  Set speed (17.1 mm/s)
  Call Extruder(548.01735)
  MoveL 6241 to (555.94, 469.94, 108) mm, rotated rx 180 ry 0 rz 160 deg; joints [2.142, 70.681, -21.623, -151.69, 52.63, 161.895]
  Set speed (17.1 mm/s)
  Call Extruder(550.98604)
  MoveL 6242 to (556.35, 470.73, 108) mm, rotated rx 180 ry 0 rz 160 deg; joints [2.23, 70.775, -21.811, -151.55, 52.574, 161.774]
  Set speed (17.1 mm/s)
  Call Extruder(555.34472)
  MoveL 6243 to (556.95, 471.91, 108) mm, rotated rx 180 ry 0 rz 160 deg; joints [2.36, 70.91, -22.084, -151.344, 52.494, 161.596]
  Set speed (17.1 mm/s)
  Call Extruder(559.57401)
  MoveL 6244 to (557.5, 473.06, 108) mm, rotated rx -180 ry 0 rz 160 deg; joints [2.488, 71.037, -22.339, -151.143, 52.422, 161.425]
  Set speed (17.1 mm/s)
  Call Extruder(563.96084)
  MoveL 6245 to (558.05, 474.27, 108) mm, rotated rx -180 ry 0 rz 160 deg; joints [2.621, 71.165, -22.597, -150.936, 52.351, 161.248]
  Set speed (17.1 mm/s)
  Call Extruder(568.24026)
  MoveL 6246 to (558.56, 475.46, 108) mm, rotated rx 180 ry 0 rz 160 deg; joints [2.752, 71.285, -22.838, -150.733, 52.288, 161.078]
  Set speed (17.1 mm/s)
  Call Extruder(572.63486)
  MoveL 6247 to (559.07, 476.69, 108) mm, rotated rx 180 ry 0 rz 160 deg; joints [2.888, 71.406, -23.081, -150.525, 52.225, 160.903]
  Set speed (17.0 mm/s)
  Call Extruder(577.61580)
  MoveL 6248 to (559.6, 478.09, 108) mm, rotated rx 180 ry 0 rz 160 deg; joints [3.043, 71.535, -23.342, -150.289, 52.162, 160.707]
  Set speed (17.0 mm/s)
  Call Extruder(581.16765)
  MoveL 6249 to (559.96, 479.1, 108) mm, rotated rx 180 ry 0 rz 160 deg; joints [3.154, 71.626, -23.524, -150.121, 52.12, 160.569]
  Set speed (17.0 mm/s)
  Call Extruder(585.42677)
  MoveL 6250 to (560.37, 480.32, 108) mm, rotated rx -180 ry 0 rz 160 deg; joints [3.288, 71.728, -23.73, -149.92, 52.075, 160.404]
  Set speed (17.1 mm/s)
  Call Extruder(589.90951)
  MoveL 6251 to (560.78, 481.61, 108) mm, rotated rx -180 ry 0 rz 160 deg; joints [3.43, 71.835, -23.944, -149.709, 52.03, 160.232]
  Set speed (17.1 mm/s)
  Call Extruder(594.01666)
  MoveL 6252 to (561.12, 482.81, 108) mm, rotated rx 180 ry 0 rz 160 deg; joints [3.561, 71.925, -24.125, -149.516, 51.996, 160.077]
  Call Extruder(598.21491)
  MoveL 6253 to (561.46, 484.03, 108) mm, rotated rx 180 ry 0 rz 160 deg; joints [3.695, 72.016, -24.307, -149.32, 51.963, 159.919]
  Set speed (17.1 mm/s)
  Call Extruder(602.61345)
  MoveL 6254 to (561.77, 485.32, 108) mm, rotated rx -180 ry 0 rz 160 deg; joints [3.837, 72.104, -24.483, -149.115, 51.936, 159.758]
  Call Extruder(606.81186)
  MoveL 6255 to (562.06, 486.56, 108) mm, rotated rx -180 ry 0 rz 160 deg; joints [3.973, 72.186, -24.648, -148.92, 51.912, 159.604]
  Set speed (17.1 mm/s)
  Call Extruder(615.47372)
  MoveL 6256 to (562.56, 489.13, 108) mm, rotated rx 180 ry 0 rz 160 deg; joints [4.256, 72.337, -24.952, -148.522, 51.881, 159.296]
  Set speed (17.1 mm/s)
  Call Extruder(624.04952)
  MoveL 6257 to (562.96, 491.7, 108) mm, rotated rx 180 ry 0 rz 160 deg; joints [4.538, 72.468, -25.214, -148.133, 51.87, 159.001]
  Call Extruder(632.73234)
  MoveL 6258 to (563.25, 494.31, 108) mm, rotated rx 180 ry 0 rz 160 deg; joints [4.825, 72.581, -25.44, -147.745, 51.877, 158.714]
  Set speed (17.1 mm/s)
  Call Extruder(641.21506)
  MoveL 6259 to (563.42, 496.87, 108) mm, rotated rx 180 ry 0 rz 160 deg; joints [5.108, 72.671, -25.62, -147.373, 51.905, 158.447]
  Call Extruder(649.80353)
  MoveL 6260 to (563.5, 499.47, 108) mm, rotated rx 180 ry 0 rz 160 deg; joints [5.395, 72.741, -25.761, -147.004, 51.951, 158.189]
  Set speed (17.1 mm/s)
  Call Extruder(658.25838)
  MoveL 6261 to (563.47, 502.03, 108) mm, rotated rx 180 ry 0 rz 160 deg; joints [5.678, 72.79, -25.859, -146.649, 52.016, 157.949]
  Set speed (17.1 mm/s)
  Call Extruder(666.94750)
  MoveL 6262 to (563.33, 504.65, 108) mm, rotated rx 180 ry 0 rz 160 deg; joints [5.97, 72.82, -25.918, -146.293, 52.102, 157.718]
  Set speed (17.1 mm/s)
  Call Extruder(675.54081)
  MoveL 6263 to (563.09, 507.24, 108) mm, rotated rx 180 ry 0 rz 160 deg; joints [6.259, 72.827, -25.933, -145.952, 52.206, 157.505]
  Set speed (17.1 mm/s)
  Call Extruder(684.21964)
  MoveL 6264 to (562.73, 509.85, 108) mm, rotated rx -180 ry 0 rz 160 deg; joints [6.552, 72.813, -25.905, -145.617, 52.329, 157.306]
  Set speed (17.1 mm/s)
  Call Extruder(692.70275)
  MoveL 6265 to (562.29, 512.38, 108) mm, rotated rx -180 ry 0 rz 160 deg; joints [6.837, 72.779, -25.837, -145.3, 52.468, 157.128]
  Set speed (17.1 mm/s)
  Call Extruder(701.33186)
  MoveL 6266 to (561.72, 514.93, 108) mm, rotated rx 180 ry 0 rz 160 deg; joints [7.126, 72.723, -25.725, -144.989, 52.627, 156.965]
  Set speed (17.1 mm/s)
  Call Extruder(705.59645)
  MoveL 6267 to (561.4, 516.17, 108) mm, rotated rx 180 ry 0 rz 160 deg; joints [7.268, 72.686, -25.651, -144.841, 52.713, 156.892]
  Set speed (17.1 mm/s)
  Call Extruder(709.78855)
  MoveL 6268 to (561.07, 517.4, 108) mm, rotated rx -180 ry 0 rz 160 deg; joints [7.408, 72.648, -25.574, -144.696, 52.799, 156.822]
  Call Extruder(714.24503)
  MoveL 6269 to (560.68, 518.69, 108) mm, rotated rx -180 ry 0 rz 160 deg; joints [7.556, 72.599, -25.476, -144.547, 52.897, 156.754]
  Set speed (17.1 mm/s)
  Call Extruder(718.50186)
  MoveL 6270 to (560.3, 519.91, 108) mm, rotated rx 180 ry 0 rz 160 deg; joints [7.697, 72.55, -25.377, -144.406, 52.994, 156.692]
  Call Extruder(722.79606)
  MoveL 6271 to (559.87, 521.14, 108) mm, rotated rx -180 ry 0 rz 160 deg; joints [7.839, 72.492, -25.263, -144.268, 53.096, 156.636]
  Set speed (17.1 mm/s)
  Call Extruder(727.21508)
  MoveL 6272 to (559.42, 522.4, 108) mm, rotated rx 180 ry 0 rz 160 deg; joints [7.985, 72.431, -25.14, -144.128, 53.204, 156.581]
  Set speed (17.1 mm/s)
  Call Extruder(731.38954)
  MoveL 6273 to (558.96, 523.57, 108) mm, rotated rx 180 ry 0 rz 160 deg; joints [8.122, 72.366, -25.009, -144, 53.312, 156.535]
  Call Extruder(735.57075)
  MoveL 6274 to (558.48, 524.74, 108) mm, rotated rx -180 ry 0 rz 160 deg; joints [8.258, 72.298, -24.874, -143.873, 53.421, 156.492]
  Set speed (17.1 mm/s)
  Call Extruder(739.97869)
  MoveL 6275 to (557.95, 525.96, 108) mm, rotated rx -180 ry 0 rz 160 deg; joints [8.402, 72.22, -24.716, -143.744, 53.542, 156.452]
  Call Extruder(744.11811)
  MoveL 6276 to (557.43, 527.1, 108) mm, rotated rx 180 ry 0 rz 160 deg; joints [8.537, 72.144, -24.564, -143.624, 53.658, 156.418]
  Set speed (17.1 mm/s)
  Call Extruder(747.32998)
  MoveL 6277 to (557.01, 527.98, 108) mm, rotated rx -180 ry 0 rz 160 deg; joints [8.64, 72.081, -24.437, -143.534, 53.75, 156.395]
  Set speed (17.1 mm/s)
  Call Extruder(752.75463)
  MoveL 6278 to (556.26, 529.44, 108) mm, rotated rx 180 ry 0 rz 160 deg; joints [8.815, 71.968, -24.212, -143.385, 53.911, 156.361]
  Set speed (17.1 mm/s)
  Call Extruder(757.06415)
  MoveL 6279 to (555.65, 530.59, 108) mm, rotated rx -180 ry 0 rz 160 deg; joints [8.953, 71.874, -24.022, -143.27, 54.043, 156.34]
  Set speed (17.1 mm/s)
  Call Extruder(761.47227)
  MoveL 6280 to (554.99, 531.75, 108) mm, rotated rx -180 ry 0 rz 160 deg; joints [9.093, 71.772, -23.818, -143.156, 54.181, 156.322]
  Set speed (17.1 mm/s)
  Call Extruder(765.64450)
  MoveL 6281 to (554.35, 532.84, 108) mm, rotated rx 180 ry 0 rz 160 deg; joints [9.225, 71.673, -23.618, -143.05, 54.314, 156.31]
  Set speed (17.1 mm/s)
  Call Extruder(769.99840)
  MoveL 6282 to (553.66, 533.96, 108) mm, rotated rx 180 ry 0 rz 160 deg; joints [9.362, 71.564, -23.399, -142.944, 54.457, 156.301]
  Set speed (17.1 mm/s)
  Call Extruder(774.22100)
  MoveL 6283 to (552.96, 535.03, 108) mm, rotated rx 180 ry 0 rz 160 deg; joints [9.494, 71.454, -23.178, -142.843, 54.599, 156.297]
  Set speed (17.1 mm/s)
  Call Extruder(778.57699)
  MoveL 6284 to (552.23, 536.12, 108) mm, rotated rx -180 ry 0 rz 160 deg; joints [9.629, 71.337, -22.943, -142.743, 54.747, 156.298]
  Set speed (17.1 mm/s)
  Call Extruder(782.79357)
  MoveL 6285 to (551.49, 537.17, 108) mm, rotated rx 180 ry 0 rz 160 deg; joints [9.758, 71.219, -22.706, -142.648, 54.894, 156.302]
  Set speed (17.1 mm/s)
  Call Extruder(787.24564)
  MoveL 6286 to (550.69, 538.25, 108) mm, rotated rx 180 ry 0 rz 160 deg; joints [9.894, 71.091, -22.448, -142.551, 55.052, 156.311]
  Set speed (17.1 mm/s)
  Call Extruder(791.44936)
  MoveL 6287 to (549.91, 539.26, 108) mm, rotated rx 180 ry 0 rz 160 deg; joints [10.021, 70.966, -22.196, -142.463, 55.204, 156.324]
  Set speed (17.1 mm/s)
  Call Extruder(795.66917)
  MoveL 6288 to (549.11, 540.25, 108) mm, rotated rx -180 ry 0 rz 160 deg; joints [10.148, 70.837, -21.937, -142.377, 55.358, 156.34]
  Set speed (17.1 mm/s)
  Call Extruder(799.97665)
  MoveL 6289 to (548.28, 541.25, 108) mm, rotated rx 180 ry 0 rz 160 deg; joints [10.277, 70.702, -21.664, -142.292, 55.518, 156.362]
  Call Extruder(804.28620)
  MoveL 6290 to (547.42, 542.24, 108) mm, rotated rx 180 ry 0 rz 160 deg; joints [10.404, 70.563, -21.383, -142.211, 55.681, 156.387]
  Set speed (17.1 mm/s)
  Call Extruder(808.67868)
  MoveL 6291 to (546.52, 543.22, 108) mm, rotated rx 180 ry 0 rz 160 deg; joints [10.532, 70.418, -21.091, -142.13, 55.849, 156.416]
  Set speed (17.1 mm/s)
  Call Extruder(812.90239)
  MoveL 6292 to (545.65, 544.15, 108) mm, rotated rx 180 ry 0 rz 160 deg; joints [10.654, 70.275, -20.802, -142.055, 56.013, 156.449]
  Call Extruder(817.23909)
  MoveL 6293 to (544.72, 545.08, 108) mm, rotated rx 180 ry 0 rz 160 deg; joints [10.778, 70.124, -20.499, -141.982, 56.183, 156.486]
  Set speed (17.1 mm/s)
  Call Extruder(821.47958)
  MoveL 6294 to (543.8, 545.98, 108) mm, rotated rx -180 ry 0 rz 160 deg; joints [10.898, 69.975, -20.196, -141.912, 56.351, 156.526]
  Set speed (17.1 mm/s)
  Call Extruder(825.79664)
  MoveL 6295 to (542.85, 546.87, 108) mm, rotated rx -180 ry 0 rz 160 deg; joints [11.018, 69.819, -19.881, -141.845, 56.524, 156.571]
  Set speed (17.1 mm/s)
  Call Extruder(830.02754)
  MoveL 6296 to (541.89, 547.72, 108) mm, rotated rx 180 ry 0 rz 160 deg; joints [11.135, 69.663, -19.566, -141.781, 56.696, 156.618]
  Set speed (17.1 mm/s)
  Call Extruder(834.31470)
  MoveL 6297 to (540.91, 548.57, 108) mm, rotated rx 180 ry 0 rz 160 deg; joints [11.252, 69.503, -19.241, -141.72, 56.871, 156.669]
  Set speed (17.1 mm/s)
  Call Extruder(838.61022)
  MoveL 6298 to (539.91, 549.39, 108) mm, rotated rx -180 ry 0 rz 160 deg; joints [11.368, 69.339, -18.91, -141.661, 57.048, 156.724]
  Call Extruder(842.95745)
  MoveL 6299 to (538.88, 550.21, 108) mm, rotated rx 180 ry 0 rz 160 deg; joints [11.483, 69.171, -18.569, -141.604, 57.229, 156.783]
  Set speed (17.1 mm/s)
  Call Extruder(847.19189)
  MoveL 6300 to (537.86, 550.98, 108) mm, rotated rx -180 ry 0 rz 160 deg; joints [11.594, 69.004, -18.232, -141.551, 57.407, 156.844]
  Call Extruder(851.49280)
  MoveL 6301 to (536.8, 551.75, 108) mm, rotated rx -180 ry 0 rz 160 deg; joints [11.705, 68.833, -17.884, -141.5, 57.589, 156.909]
  Set speed (17.1 mm/s)
  Call Extruder(855.84391)
  MoveL 6302 to (535.72, 552.5, 108) mm, rotated rx 180 ry 0 rz 160 deg; joints [11.815, 68.657, -17.526, -141.451, 57.774, 156.978]
  Call Extruder(860.13738)
  MoveL 6303 to (534.64, 553.22, 108) mm, rotated rx 180 ry 0 rz 160 deg; joints [11.922, 68.481, -17.169, -141.406, 57.958, 157.05]
  Set speed (17.1 mm/s)
  Call Extruder(864.36320)
  MoveL 6304 to (533.56, 553.91, 108) mm, rotated rx 180 ry 0 rz 160 deg; joints [12.026, 68.305, -16.812, -141.363, 58.14, 157.124]
  Call Extruder(868.65744)
  MoveL 6305 to (532.46, 554.58, 108) mm, rotated rx 180 ry 0 rz 160 deg; joints [12.13, 68.125, -16.446, -141.323, 58.325, 157.201]
  Set speed (17.1 mm/s)
  Call Extruder(872.95693)
  MoveL 6306 to (531.33, 555.24, 108) mm, rotated rx -180 ry 0 rz 160 deg; joints [12.232, 67.942, -16.073, -141.285, 58.513, 157.282]
  Set speed (17.1 mm/s)
  Call Extruder(877.46939)
  MoveL 6307 to (530.13, 555.9, 108) mm, rotated rx 180 ry 0 rz 160 deg; joints [12.337, 67.748, -15.679, -141.248, 58.71, 157.37]
  Set speed (17.1 mm/s)
  Call Extruder(882.84168)
  MoveL 6308 to (528.69, 556.65, 108) mm, rotated rx -180 ry 0 rz 160 deg; joints [12.459, 67.516, -15.204, -141.208, 58.945, 157.479]
  Set speed (17.1 mm/s)
  Call Extruder(885.82668)
  MoveL 6309 to (527.89, 557.05, 108) mm, rotated rx 180 ry 0 rz 160 deg; joints [12.525, 67.385, -14.937, -141.188, 59.077, 157.542]
  Set speed (17.1 mm/s)
  Call Extruder(890.27350)
  MoveL 6310 to (526.67, 557.63, 108) mm, rotated rx 180 ry 0 rz 160 deg; joints [12.623, 67.188, -14.537, -141.16, 59.273, 157.637]
  Set speed (17.1 mm/s)
  Call Extruder(894.52079)
  MoveL 6311 to (525.5, 558.15, 108) mm, rotated rx 180 ry 0 rz 160 deg; joints [12.713, 66.999, -14.15, -141.136, 59.461, 157.732]
  Set speed (17.1 mm/s)
  Call Extruder(898.80163)
  MoveL 6312 to (524.31, 558.66, 108) mm, rotated rx -180 ry 0 rz 160 deg; joints [12.803, 66.808, -13.76, -141.113, 59.65, 157.828]
  Call Extruder(903.10551)
  MoveL 6313 to (523.1, 559.14, 108) mm, rotated rx 180 ry 0 rz 160 deg; joints [12.89, 66.613, -13.361, -141.095, 59.841, 157.929]
  Set speed (17.1 mm/s)
  Call Extruder(907.22766)
  MoveL 6314 to (521.94, 559.59, 108) mm, rotated rx -180 ry 0 rz 160 deg; joints [12.972, 66.427, -12.979, -141.078, 60.024, 158.027]
  Set speed (17.0 mm/s)
  Call Extruder(911.77097)
  MoveL 6315 to (520.64, 560.05, 108) mm, rotated rx 180 ry 0 rz 160 deg; joints [13.059, 66.219, -12.554, -141.063, 60.226, 158.138]
  Set speed (17.0 mm/s)
  Call Extruder(916.06108)
  MoveL 6316 to (519.42, 560.46, 108) mm, rotated rx 180 ry 0 rz 160 deg; joints [13.141, 66.023, -12.152, -141.05, 60.416, 158.244]
  Call Extruder(921.22931)
  MoveL 6317 to (517.92, 560.92, 108) mm, rotated rx 180 ry 0 rz 160 deg; joints [13.234, 65.785, -11.662, -141.039, 60.646, 158.377]
  Set speed (17.1 mm/s)
  Call Extruder(924.56731)
  MoveL 6318 to (516.96, 561.2, 108) mm, rotated rx 180 ry 0 rz 160 deg; joints [13.293, 65.63, -11.345, -141.033, 60.795, 158.463]
  Set speed (17.1 mm/s)
  Call Extruder(928.35137)
  MoveL 6319 to (515.85, 561.49, 108) mm, rotated rx -180 ry 0 rz 160 deg; joints [13.358, 65.454, -10.983, -141.03, 60.963, 158.564]
  Set speed (17.0 mm/s)
  Call Extruder(933.06141)
  MoveL 6320 to (514.47, 561.83, 108) mm, rotated rx -180 ry 0 rz 160 deg; joints [13.436, 65.235, -10.531, -141.027, 61.172, 158.69]
  Set speed (17.1 mm/s)
  Call Extruder(941.79542)
  MoveL 6321 to (511.88, 562.38, 108) mm, rotated rx 180 ry 0 rz 160 deg; joints [13.573, 64.825, -9.687, -141.031, 61.559, 158.932]
  Call Extruder(950.43348)
  MoveL 6322 to (509.31, 562.82, 108) mm, rotated rx 180 ry 0 rz 160 deg; joints [13.698, 64.417, -8.846, -141.045, 61.941, 159.179]
  Set speed (17.1 mm/s)
  Call Extruder(958.92783)
  MoveL 6323 to (506.76, 563.14, 108) mm, rotated rx 180 ry 0 rz 160 deg; joints [13.81, 64.015, -8.015, -141.069, 62.315, 159.428]
  Call Extruder(967.57110)
  MoveL 6324 to (504.15, 563.37, 108) mm, rotated rx 180 ry 0 rz 160 deg; joints [13.913, 63.606, -7.166, -141.104, 62.692, 159.689]
  Set speed (17.1 mm/s)
  Call Extruder(976.19607)
  MoveL 6325 to (501.54, 563.48, 108) mm, rotated rx -180 ry 0 rz 160 deg; joints [14.005, 63.197, -6.319, -141.148, 63.065, 159.954]
  Set speed (17.1 mm/s)
  Call Extruder(984.68341)
  MoveL 6326 to (498.98, 563.49, 108) mm, rotated rx -180 ry 0 rz 160 deg; joints [14.083, 62.796, -5.484, -141.203, 63.43, 160.222]
  Set speed (10.0 mm/s)
  MoveL 6327 to (498.98, 563.49, 112) mm, rotated rx 180 ry 0 rz 160 deg; joints [14.083, 62.174, -5.222, -141.089, 63.149, 159.969]
  Set speed (120.0 mm/s)
  MoveL 6328 to (499.03, 561.95, 112) mm, rotated rx 180 ry 0 rz 160 deg; joints [13.896, 62.122, -5.115, -141.304, 63.129, 160.097]
  Set speed (16.5 mm/s)
  Call Extruder(993.61366)
  MoveL 6329 to (496.42, 561.86, 112) mm, rotated rx 180 ry 0 rz 160 deg; joints [13.962, 61.713, -4.268, -141.371, 63.493, 160.371]
  Set speed (16.5 mm/s)
  Call Extruder(1002.30166)
  MoveL 6330 to (493.88, 561.66, 112) mm, rotated rx 180 ry 0 rz 160 deg; joints [14.015, 61.317, -3.446, -141.448, 63.844, 160.643]
  Call Extruder(1010.77384)
  MoveL 6331 to (491.42, 561.36, 112) mm, rotated rx 180 ry 0 rz 160 deg; joints [14.054, 60.933, -2.647, -141.532, 64.181, 160.913]
  Set speed (16.5 mm/s)
  Call Extruder(1019.51677)
  MoveL 6332 to (488.89, 560.96, 112) mm, rotated rx 180 ry 0 rz 160 deg; joints [14.082, 60.539, -1.827, -141.63, 64.524, 161.194]
  Set speed (16.5 mm/s)
  Call Extruder(1028.25434)
  MoveL 6333 to (486.38, 560.45, 112) mm, rotated rx 180 ry 0 rz 160 deg; joints [14.096, 60.149, -1.014, -141.739, 64.861, 161.478]
  Set speed (16.5 mm/s)
  Call Extruder(1036.68997)
  MoveL 6334 to (483.99, 559.86, 112) mm, rotated rx -180 ry 0 rz 160 deg; joints [14.098, 59.777, -0.235, -141.855, 65.181, 161.754]
  Set speed (16.5 mm/s)
  Call Extruder(1041.17353)
  MoveL 6335 to (482.73, 559.5, 112) mm, rotated rx 180 ry 0 rz 160 deg; joints [14.093, 59.581, 0.176, -141.921, 65.348, 161.902]
  Call Extruder(1045.35326)
  MoveL 6336 to (481.56, 559.15, 112) mm, rotated rx 180 ry 0 rz 160 deg; joints [14.086, 59.399, 0.557, -141.984, 65.503, 162.04]
  Call Extruder(1049.82255)
  MoveL 6337 to (480.31, 558.74, 112) mm, rotated rx -180 ry 0 rz 160 deg; joints [14.074, 59.206, 0.962, -142.056, 65.666, 162.189]
  Set speed (16.5 mm/s)
  Call Extruder(1053.93208)
  MoveL 6338 to (479.18, 558.35, 112) mm, rotated rx -180 ry 0 rz 160 deg; joints [14.061, 59.03, 1.333, -142.123, 65.816, 162.325]
  Set speed (16.5 mm/s)
  Call Extruder(1058.54264)
  MoveL 6339 to (477.91, 557.88, 112) mm, rotated rx -180 ry 0 rz 160 deg; joints [14.041, 58.833, 1.745, -142.203, 65.981, 162.479]
  Set speed (16.5 mm/s)
  Call Extruder(1062.60609)
  MoveL 6340 to (476.81, 557.46, 112) mm, rotated rx 180 ry 0 rz 160 deg; joints [14.022, 58.662, 2.107, -142.275, 66.125, 162.614]
  Set speed (16.5 mm/s)
  Call Extruder(1065.13276)
  MoveL 6341 to (476.12, 557.17, 112) mm, rotated rx 180 ry 0 rz 160 deg; joints [14.009, 58.556, 2.33, -142.321, 66.214, 162.699]
  Set speed (16.5 mm/s)
  Call Extruder(1071.22492)
  MoveL 6342 to (474.49, 556.46, 112) mm, rotated rx -180 ry 0 rz 160 deg; joints [13.97, 58.302, 2.865, -142.437, 66.425, 162.902]
  Set speed (16.5 mm/s)
  Call Extruder(1075.68538)
  MoveL 6343 to (473.31, 555.91, 112) mm, rotated rx 180 ry 0 rz 160 deg; joints [13.937, 58.118, 3.254, -142.525, 66.578, 163.052]
  Call Extruder(1080.16539)
  MoveL 6344 to (472.13, 555.34, 112) mm, rotated rx -180 ry 0 rz 160 deg; joints [13.901, 57.935, 3.641, -142.616, 66.729, 163.202]
  Set speed (16.5 mm/s)
  Call Extruder(1083.27199)
  MoveL 6345 to (471.32, 554.93, 112) mm, rotated rx -180 ry 0 rz 160 deg; joints [13.874, 57.809, 3.907, -142.681, 66.833, 163.305]
  Set speed (16.5 mm/s)
  Call Extruder(1088.62781)
  MoveL 6346 to (469.94, 554.18, 112) mm, rotated rx -180 ry 0 rz 160 deg; joints [13.822, 57.594, 4.362, -142.797, 67.009, 163.484]
  Set speed (16.5 mm/s)
  Call Extruder(1093.83533)
  MoveL 6347 to (468.62, 553.42, 112) mm, rotated rx 180 ry 0 rz 160 deg; joints [13.766, 57.388, 4.798, -142.914, 67.177, 163.658]
  Set speed (16.5 mm/s)
  Call Extruder(1096.84420)
  MoveL 6348 to (467.86, 552.97, 112) mm, rotated rx -180 ry 0 rz 160 deg; joints [13.731, 57.27, 5.049, -142.983, 67.273, 163.759]
  Set speed (16.5 mm/s)
  Call Extruder(1101.63964)
  MoveL 6349 to (466.67, 552.23, 112) mm, rotated rx 180 ry 0 rz 160 deg; joints [13.673, 57.084, 5.444, -143.097, 67.424, 163.919]
  Set speed (16.5 mm/s)
  Call Extruder(1106.16464)
  MoveL 6350 to (465.56, 551.51, 112) mm, rotated rx 180 ry 0 rz 160 deg; joints [13.614, 56.911, 5.812, -143.207, 67.563, 164.069]
  Call Extruder(1110.49447)
  MoveL 6351 to (464.51, 550.79, 112) mm, rotated rx 180 ry 0 rz 160 deg; joints [13.553, 56.747, 6.161, -143.315, 67.695, 164.212]
  Call Extruder(1114.72597)
  MoveL 6352 to (463.51, 550.07, 112) mm, rotated rx 180 ry 0 rz 160 deg; joints [13.491, 56.589, 6.497, -143.424, 67.821, 164.352]
  Set speed (16.5 mm/s)
  Call Extruder(1119.16395)
  MoveL 6353 to (462.46, 549.3, 112) mm, rotated rx 180 ry 0 rz 160 deg; joints [13.421, 56.426, 6.846, -143.541, 67.952, 164.498]
  Set speed (16.5 mm/s)
  Call Extruder(1123.30803)
  MoveL 6354 to (461.5, 548.55, 112) mm, rotated rx 180 ry 0 rz 160 deg; joints [13.353, 56.275, 7.167, -143.652, 68.071, 164.634]
  Call Extruder(1127.16809)
  MoveL 6355 to (460.63, 547.84, 112) mm, rotated rx 180 ry 0 rz 160 deg; joints [13.287, 56.137, 7.463, -143.759, 68.18, 164.76]
  Set speed (16.5 mm/s)
  Call Extruder(1131.97091)
  MoveL 6356 to (459.55, 546.94, 112) mm, rotated rx 180 ry 0 rz 160 deg; joints [13.2, 55.967, 7.826, -143.894, 68.314, 164.916]
  Set speed (16.5 mm/s)
  Call Extruder(1135.81592)
  MoveL 6357 to (458.7, 546.19, 112) mm, rotated rx -180 ry 0 rz 160 deg; joints [13.128, 55.834, 8.112, -144.005, 68.418, 165.04]
  Set speed (16.5 mm/s)
  Call Extruder(1140.08255)
  MoveL 6358 to (457.78, 545.35, 112) mm, rotated rx -180 ry 0 rz 160 deg; joints [13.044, 55.688, 8.425, -144.131, 68.532, 165.178]
  Set speed (16.5 mm/s)
  Call Extruder(1144.40860)
  MoveL 6359 to (456.86, 544.48, 112) mm, rotated rx 180 ry 0 rz 160 deg; joints [12.956, 55.542, 8.737, -144.261, 68.645, 165.316]
  Set speed (16.5 mm/s)
  Call Extruder(1149.46065)
  MoveL 6360 to (455.82, 543.44, 112) mm, rotated rx 180 ry 0 rz 160 deg; joints [12.848, 55.375, 9.095, -144.416, 68.773, 165.476]
  Set speed (16.5 mm/s)
  Call Extruder(1153.62057)
  MoveL 6361 to (454.97, 542.56, 112) mm, rotated rx 180 ry 0 rz 160 deg; joints [12.756, 55.24, 9.386, -144.546, 68.876, 165.608]
  Set speed (16.5 mm/s)
  Call Extruder(1157.48411)
  MoveL 6362 to (454.2, 541.73, 112) mm, rotated rx -180 ry 0 rz 160 deg; joints [12.668, 55.118, 9.65, -144.67, 68.97, 165.729]
  Set speed (16.5 mm/s)
  Call Extruder(1162.79369)
  MoveL 6363 to (453.17, 540.57, 112) mm, rotated rx 180 ry 0 rz 160 deg; joints [12.542, 54.952, 10.008, -144.843, 69.096, 165.894]
  Set speed (16.5 mm/s)
  Call Extruder(1166.69723)
  MoveL 6364 to (452.43, 539.7, 112) mm, rotated rx 180 ry 0 rz 160 deg; joints [12.445, 54.833, 10.264, -144.973, 69.185, 166.014]
  Set speed (16.5 mm/s)
  Call Extruder(1170.90886)
  MoveL 6365 to (451.65, 538.75, 112) mm, rotated rx 180 ry 0 rz 160 deg; joints [12.339, 54.706, 10.537, -145.116, 69.279, 166.143]
  Call Extruder(1175.28579)
  MoveL 6366 to (450.86, 537.74, 112) mm, rotated rx 180 ry 0 rz 160 deg; joints [12.225, 54.578, 10.814, -145.266, 69.374, 166.276]
  Set speed (16.5 mm/s)
  Call Extruder(1179.12057)
  MoveL 6367 to (450.18, 536.84, 112) mm, rotated rx 180 ry 0 rz 160 deg; joints [12.122, 54.468, 11.052, -145.401, 69.455, 166.391]
  Call Extruder(1183.36849)
  MoveL 6368 to (449.45, 535.83, 112) mm, rotated rx -180 ry 0 rz 160 deg; joints [12.005, 54.349, 11.31, -145.551, 69.542, 166.517]
  Call Extruder(1188.42759)
  MoveL 6369 to (448.61, 534.61, 112) mm, rotated rx 180 ry 0 rz 160 deg; joints [11.862, 54.21, 11.61, -145.734, 69.642, 166.666]
  Call Extruder(1192.74712)
  MoveL 6370 to (447.91, 533.56, 112) mm, rotated rx -180 ry 0 rz 160 deg; joints [11.736, 54.095, 11.86, -145.892, 69.725, 166.792]
  Call Extruder(1196.57342)
  MoveL 6371 to (447.32, 532.61, 112) mm, rotated rx 180 ry 0 rz 160 deg; joints [11.622, 53.996, 12.075, -146.035, 69.795, 166.903]
  Set speed (16.5 mm/s)
  Call Extruder(1201.40136)
  MoveL 6372 to (446.59, 531.4, 112) mm, rotated rx -180 ry 0 rz 160 deg; joints [11.475, 53.874, 12.341, -146.217, 69.881, 167.04]
  Set speed (16.5 mm/s)
  Call Extruder(1205.58846)
  MoveL 6373 to (445.98, 530.34, 112) mm, rotated rx 180 ry 0 rz 160 deg; joints [11.344, 53.771, 12.564, -146.377, 69.952, 167.158]
  Set speed (16.5 mm/s)
  Call Extruder(1210.01458)
  MoveL 6374 to (445.35, 529.2, 112) mm, rotated rx 180 ry 0 rz 160 deg; joints [11.203, 53.665, 12.794, -146.548, 70.024, 167.281]
  Set speed (16.5 mm/s)
  Call Extruder(1215.95240)
  MoveL 6375 to (444.55, 527.66, 112) mm, rotated rx 180 ry 0 rz 160 deg; joints [11.009, 53.529, 13.092, -146.782, 70.116, 167.444]
  Set speed (16.5 mm/s)
  Call Extruder(1218.75277)
  MoveL 6376 to (444.19, 526.92, 112) mm, rotated rx 180 ry 0 rz 160 deg; joints [10.915, 53.467, 13.227, -146.894, 70.157, 167.52]
  Set speed (16.5 mm/s)
  Call Extruder(1223.04451)
  MoveL 6377 to (443.66, 525.78, 112) mm, rotated rx 180 ry 0 rz 160 deg; joints [10.769, 53.375, 13.428, -147.067, 70.217, 167.634]
  Set speed (16.5 mm/s)
  Call Extruder(1227.26126)
  MoveL 6378 to (443.16, 524.66, 112) mm, rotated rx -180 ry 0 rz 160 deg; joints [10.624, 53.286, 13.621, -147.237, 70.274, 167.745]
  Call Extruder(1231.72537)
  MoveL 6379 to (442.65, 523.45, 112) mm, rotated rx 180 ry 0 rz 160 deg; joints [10.467, 53.197, 13.816, -147.421, 70.33, 167.861]
  Set speed (16.5 mm/s)
  Call Extruder(1235.77011)
  MoveL 6380 to (442.21, 522.36, 112) mm, rotated rx 180 ry 0 rz 160 deg; joints [10.323, 53.118, 13.988, -147.588, 70.379, 167.964]
  Set speed (16.5 mm/s)
  Call Extruder(1240.37793)
  MoveL 6381 to (441.75, 521.09, 112) mm, rotated rx -180 ry 0 rz 160 deg; joints [10.156, 53.033, 14.174, -147.781, 70.429, 168.08]
  Call Extruder(1244.73243)
  MoveL 6382 to (441.32, 519.89, 112) mm, rotated rx 180 ry 0 rz 160 deg; joints [9.997, 52.955, 14.346, -147.964, 70.475, 168.188]
  Set speed (16.5 mm/s)
  Call Extruder(1249.05341)
  MoveL 6383 to (440.93, 518.69, 112) mm, rotated rx -180 ry 0 rz 160 deg; joints [9.835, 52.882, 14.506, -148.148, 70.516, 168.293]
  Set speed (16.5 mm/s)
  Call Extruder(1253.21630)
  MoveL 6384 to (440.57, 517.53, 112) mm, rotated rx -180 ry 0 rz 160 deg; joints [9.678, 52.813, 14.656, -148.326, 70.554, 168.393]
  Set speed (16.5 mm/s)
  Call Extruder(1261.92076)
  MoveL 6385 to (439.9, 515.07, 112) mm, rotated rx -180 ry 0 rz 160 deg; joints [9.342, 52.682, 14.944, -148.704, 70.621, 168.596]
  Set speed (16.5 mm/s)
  Call Extruder(1266.37934)
  MoveL 6386 to (439.6, 513.8, 112) mm, rotated rx -180 ry 0 rz 160 deg; joints [9.167, 52.62, 15.079, -148.899, 70.649, 168.696]
  Call Extruder(1270.50108)
  MoveL 6387 to (439.34, 512.63, 112) mm, rotated rx 180 ry 0 rz 160 deg; joints [9.004, 52.566, 15.198, -149.081, 70.673, 168.788]
  Set speed (16.5 mm/s)
  Call Extruder(1279.45107)
  MoveL 6388 to (438.86, 510.05, 112) mm, rotated rx 180 ry 0 rz 160 deg; joints [8.644, 52.459, 15.433, -149.478, 70.713, 168.981]
  Call Extruder(1288.11358)
  MoveL 6389 to (438.5, 507.54, 112) mm, rotated rx 180 ry 0 rz 160 deg; joints [8.289, 52.371, 15.627, -149.866, 70.738, 169.159]
  Set speed (16.5 mm/s)
  Call Extruder(1296.77064)
  MoveL 6390 to (438.24, 505.02, 112) mm, rotated rx 180 ry 0 rz 160 deg; joints [7.929, 52.296, 15.792, -150.256, 70.748, 169.33]
  Set speed (16.5 mm/s)
  Call Extruder(1305.30799)
  MoveL 6391 to (438.09, 502.52, 112) mm, rotated rx 180 ry 0 rz 160 deg; joints [7.57, 52.237, 15.922, -150.642, 70.744, 169.491]
  Set speed (16.5 mm/s)
  Call Extruder(1313.89422)
  MoveL 6392 to (438.04, 500.01, 112) mm, rotated rx -180 ry 0 rz 160 deg; joints [7.205, 52.192, 16.022, -151.032, 70.726, 169.644]
  Call Extruder(1321.77669)
  MoveL 6393 to (438.08, 497.7, 112) mm, rotated rx -180 ry 0 rz 160 deg; joints [6.868, 52.162, 16.086, -151.389, 70.697, 169.778]
  Set speed (16.5 mm/s)
  Call Extruder(1329.55299)
  MoveL 6394 to (438.21, 495.43, 112) mm, rotated rx 180 ry 0 rz 160 deg; joints [6.535, 52.145, 16.124, -151.74, 70.656, 169.904]
  Set speed (16.5 mm/s)
  Call Extruder(1337.34270)
  MoveL 6395 to (438.42, 493.16, 112) mm, rotated rx 180 ry 0 rz 160 deg; joints [6.2, 52.14, 16.135, -152.091, 70.603, 170.023]
  Set speed (16.5 mm/s)
  Call Extruder(1345.13182)
  MoveL 6396 to (438.71, 490.9, 112) mm, rotated rx -180 ry 0 rz 160 deg; joints [5.865, 52.147, 16.121, -152.44, 70.538, 170.136]
  Set speed (16.5 mm/s)
  Call Extruder(1353.01280)
  MoveL 6397 to (439.09, 488.62, 112) mm, rotated rx 180 ry 0 rz 160 deg; joints [5.526, 52.165, 16.08, -152.79, 70.461, 170.243]
  Set speed (16.5 mm/s)
  Call Extruder(1360.71997)
  MoveL 6398 to (439.55, 486.41, 112) mm, rotated rx -180 ry 0 rz 160 deg; joints [5.197, 52.195, 16.014, -153.128, 70.373, 170.341]
  Set speed (16.5 mm/s)
  Call Extruder(1368.23928)
  MoveL 6399 to (440.07, 484.27, 112) mm, rotated rx -180 ry 0 rz 160 deg; joints [4.878, 52.236, 15.925, -153.454, 70.276, 170.43]
  Set speed (16.5 mm/s)
  Call Extruder(1376.30669)
  MoveL 6400 to (440.71, 482, 112) mm, rotated rx 180 ry 0 rz 160 deg; joints [4.539, 52.291, 15.804, -153.8, 70.161, 170.519]
  Call Extruder(1384.09219)
  MoveL 6401 to (441.41, 479.83, 112) mm, rotated rx -180 ry 0 rz 160 deg; joints [4.214, 52.356, 15.66, -154.127, 70.037, 170.598]
  Set speed (16.5 mm/s)
  Call Extruder(1391.88635)
  MoveL 6402 to (442.2, 477.69, 112) mm, rotated rx -180 ry 0 rz 160 deg; joints [3.894, 52.433, 15.491, -154.45, 69.902, 170.671]
  Set speed (16.5 mm/s)
  Call Extruder(1399.74827)
  MoveL 6403 to (443.06, 475.56, 112) mm, rotated rx 180 ry 0 rz 160 deg; joints [3.575, 52.522, 15.295, -154.768, 69.754, 170.738]
  Set speed (16.5 mm/s)
  Call Extruder(1407.56836)
  MoveL 6404 to (444.01, 473.47, 112) mm, rotated rx -180 ry 0 rz 160 deg; joints [3.264, 52.622, 15.076, -155.077, 69.596, 170.798]
  Set speed (16.5 mm/s)
  Call Extruder(1415.25073)
  MoveL 6405 to (445.01, 471.46, 112) mm, rotated rx -180 ry 0 rz 160 deg; joints [2.964, 52.731, 14.835, -155.372, 69.429, 170.85]
  Call Extruder(1423.15007)
  MoveL 6406 to (446.11, 469.43, 112) mm, rotated rx -180 ry 0 rz 160 deg; joints [2.662, 52.855, 14.564, -155.668, 69.247, 170.897]
  Set speed (16.5 mm/s)
  Call Extruder(1430.84754)
  MoveL 6407 to (447.26, 467.49, 112) mm, rotated rx -180 ry 0 rz 160 deg; joints [2.375, 52.986, 14.276, -155.947, 69.059, 170.936]
  Set speed (16.5 mm/s)
  Call Extruder(1438.65167)
  MoveL 6408 to (448.49, 465.56, 112) mm, rotated rx -180 ry 0 rz 160 deg; joints [2.091, 53.131, 13.961, -156.221, 68.857, 170.97]
  Set speed (16.5 mm/s)
  Call Extruder(1446.44189)
  MoveL 6409 to (449.79, 463.69, 112) mm, rotated rx 180 ry 0 rz 160 deg; joints [1.815, 53.285, 13.623, -156.484, 68.647, 170.997]
  Set speed (16.5 mm/s)
  Call Extruder(1454.32693)
  MoveL 6410 to (451.18, 461.85, 112) mm, rotated rx 180 ry 0 rz 160 deg; joints [1.545, 53.452, 13.259, -156.74, 68.423, 171.017]
  Set speed (16.5 mm/s)
  Call Extruder(1462.19959)
  MoveL 6411 to (452.63, 460.06, 112) mm, rotated rx -180 ry 0 rz 160 deg; joints [1.285, 53.63, 12.872, -156.984, 68.19, 171.031]
  Set speed (16.5 mm/s)
  Call Extruder(1469.56879)
  MoveL 6412 to (454.05, 458.44, 112) mm, rotated rx -180 ry 0 rz 160 deg; joints [1.05, 53.805, 12.489, -157.202, 67.963, 171.038]
  Set speed (16.5 mm/s)
  Call Extruder(1477.67816)
  MoveL 6413 to (455.68, 456.71, 112) mm, rotated rx 180 ry 0 rz 160 deg; joints [0.801, 54.009, 12.048, -157.43, 67.704, 171.039]
  Set speed (16.5 mm/s)
  Call Extruder(1485.39860)
  MoveL 6414 to (457.29, 455.12, 112) mm, rotated rx -180 ry 0 rz 160 deg; joints [0.574, 54.212, 11.606, -157.634, 67.449, 171.033]
  Set speed (16.5 mm/s)
  Call Extruder(1493.19948)
  MoveL 6415 to (458.97, 453.57, 112) mm, rotated rx 180 ry 0 rz 160 deg; joints [0.355, 54.427, 11.14, -157.829, 67.183, 171.02]
  Set speed (16.5 mm/s)
  Call Extruder(1501.08603)
  MoveL 6416 to (460.73, 452.08, 112) mm, rotated rx 180 ry 0 rz 160 deg; joints [0.145, 54.654, 10.649, -158.013, 66.905, 171]
  Set speed (16.5 mm/s)
  Call Extruder(1509.12428)
  MoveL 6417 to (462.57, 450.62, 112) mm, rotated rx 180 ry 0 rz 160 deg; joints [-0.059, 54.895, 10.129, -158.187, 66.615, 170.973]
  Call Extruder(1516.65650)
  MoveL 6418 to (464.36, 449.32, 112) mm, rotated rx -180 ry 0 rz 160 deg; joints [-0.239, 55.129, 9.624, -158.337, 66.335, 170.941]
  Set speed (16.5 mm/s)
  Call Extruder(1524.41183)
  MoveL 6419 to (466.24, 448.05, 112) mm, rotated rx 180 ry 0 rz 160 deg; joints [-0.413, 55.379, 9.088, -158.479, 66.04, 170.902]
  Set speed (16.5 mm/s)
  Call Extruder(1532.25228)
  MoveL 6420 to (468.18, 446.84, 112) mm, rotated rx 180 ry 0 rz 160 deg; joints [-0.578, 55.64, 8.528, -158.608, 65.736, 170.855]
  Call Extruder(1540.04391)
  MoveL 6421 to (470.16, 445.7, 112) mm, rotated rx 180 ry 0 rz 160 deg; joints [-0.73, 55.907, 7.955, -158.722, 65.427, 170.801]
  Set speed (16.5 mm/s)
  Call Extruder(1548.72627)
  MoveL 6422 to (472.41, 444.52, 112) mm, rotated rx -180 ry 0 rz 160 deg; joints [-0.886, 56.213, 7.3, -158.834, 65.077, 170.733]
  Call Extruder(1555.33105)
  MoveL 6423 to (474.15, 443.69, 112) mm, rotated rx 180 ry 0 rz 160 deg; joints [-0.995, 56.452, 6.789, -158.906, 64.806, 170.675]
  Set speed (16.5 mm/s)
  Call Extruder(1563.41114)
  MoveL 6424 to (476.32, 442.75, 112) mm, rotated rx 180 ry 0 rz 160 deg; joints [-1.117, 56.752, 6.15, -158.982, 64.469, 170.597]
  Call Extruder(1571.12783)
  MoveL 6425 to (478.42, 441.92, 112) mm, rotated rx -180 ry 0 rz 160 deg; joints [-1.222, 57.046, 5.526, -159.04, 64.143, 170.516]
  Call Extruder(0.00000)
  Set speed (16.5 mm/s)
  Call Extruder(7.86644)
  MoveL 6426 to (480.6, 441.16, 112) mm, rotated rx -180 ry 0 rz 160 deg; joints [-1.317, 57.351, 4.877, -159.085, 63.807, 170.425]
  Call Extruder(15.58996)
  MoveL 6427 to (482.76, 440.49, 112) mm, rotated rx 180 ry 0 rz 160 deg; joints [-1.399, 57.657, 4.228, -159.115, 63.473, 170.329]
  Set speed (16.5 mm/s)
  Call Extruder(23.37337)
  MoveL 6428 to (484.96, 439.9, 112) mm, rotated rx -180 ry 0 rz 160 deg; joints [-1.471, 57.971, 3.563, -159.13, 63.133, 170.224]
  Call Extruder(31.25300)
  MoveL 6429 to (487.2, 439.38, 112) mm, rotated rx -180 ry 0 rz 160 deg; joints [-1.531, 58.295, 2.879, -159.131, 62.786, 170.11]
  Set speed (16.5 mm/s)
  Call Extruder(38.96327)
  MoveL 6430 to (489.42, 438.95, 112) mm, rotated rx -180 ry 0 rz 160 deg; joints [-1.579, 58.617, 2.2, -159.119, 62.444, 169.992]
  Call Extruder(46.80296)
  MoveL 6431 to (491.69, 438.6, 112) mm, rotated rx 180 ry 0 rz 160 deg; joints [-1.616, 58.95, 1.501, -159.092, 62.095, 169.863]
  Set speed (16.5 mm/s)
  Call Extruder(54.58682)
  MoveL 6432 to (493.95, 438.34, 112) mm, rotated rx 180 ry 0 rz 160 deg; joints [-1.642, 59.284, 0.799, -159.05, 61.747, 169.728]
  Set speed (16.5 mm/s)
  Call Extruder(62.33113)
  MoveL 6433 to (496.21, 438.16, 112) mm, rotated rx -180 ry 0 rz 160 deg; joints [-1.657, 59.621, 0.093, -158.995, 61.399, 169.585]
  Set speed (16.5 mm/s)
  Call Extruder(70.20726)
  MoveL 6434 to (498.52, 438.06, 112) mm, rotated rx -180 ry 0 rz 160 deg; joints [-1.661, 59.967, -0.632, -158.925, 61.045, 169.432]
  Set speed (16.5 mm/s)
  Call Extruder(77.66521)
  MoveL 6435 to (500.7, 438.04, 112) mm, rotated rx 180 ry 0 rz 160 deg; joints [-1.655, 60.298, -1.324, -158.846, 60.71, 169.28]
  Set speed (16.5 mm/s)
  Call Extruder(85.79420)
  MoveL 6436 to (503.08, 438.12, 112) mm, rotated rx -180 ry 0 rz 160 deg; joints [-1.637, 60.662, -2.083, -158.745, 60.345, 169.106]
  Set speed (16.5 mm/s)
  Call Extruder(93.50369)
  MoveL 6437 to (505.33, 438.27, 112) mm, rotated rx -180 ry 0 rz 160 deg; joints [-1.609, 61.01, -2.807, -158.635, 60, 168.933]
  Call Extruder(101.37270)
  MoveL 6438 to (507.62, 438.51, 112) mm, rotated rx -180 ry 0 rz 160 deg; joints [-1.571, 61.367, -3.55, -158.51, 59.648, 168.748]
  Set speed (16.5 mm/s)
  Call Extruder(109.06264)
  MoveL 6439 to (509.85, 438.83, 112) mm, rotated rx -180 ry 0 rz 160 deg; joints [-1.524, 61.718, -4.278, -158.374, 59.307, 168.56]
  Call Extruder(116.96786)
  MoveL 6440 to (512.13, 439.24, 112) mm, rotated rx -180 ry 0 rz 160 deg; joints [-1.465, 62.08, -5.028, -158.222, 58.958, 168.359]
  Call Extruder(124.68471)
  MoveL 6441 to (514.34, 439.72, 112) mm, rotated rx -180 ry 0 rz 160 deg; joints [-1.399, 62.434, -5.76, -158.06, 58.621, 168.154]
  Set speed (16.5 mm/s)
  Call Extruder(132.62002)
  MoveL 6442 to (516.59, 440.3, 112) mm, rotated rx -180 ry 0 rz 160 deg; joints [-1.321, 62.799, -6.513, -157.882, 58.277, 167.937]
  Set speed (16.5 mm/s)
  Call Extruder(140.00244)
  MoveL 6443 to (518.66, 440.92, 112) mm, rotated rx -180 ry 0 rz 160 deg; joints [-1.239, 63.138, -7.213, -157.703, 57.96, 167.727]
  Set speed (16.5 mm/s)
  Call Extruder(148.11960)
  MoveL 6444 to (520.91, 441.68, 112) mm, rotated rx -180 ry 0 rz 160 deg; joints [-1.141, 63.511, -7.98, -157.495, 57.617, 167.489]
  Call Extruder(155.52464)
  MoveL 6445 to (522.94, 442.45, 112) mm, rotated rx 180 ry 0 rz 160 deg; joints [-1.043, 63.85, -8.678, -157.294, 57.307, 167.264]
  Set speed (16.5 mm/s)
  Call Extruder(163.43085)
  MoveL 6446 to (525.08, 443.34, 112) mm, rotated rx 180 ry 0 rz 160 deg; joints [-0.93, 64.211, -9.419, -157.067, 56.982, 167.018]
  Set speed (16.5 mm/s)
  Call Extruder(171.14455)
  MoveL 6447 to (527.12, 444.29, 112) mm, rotated rx -180 ry 0 rz 160 deg; joints [-0.812, 64.562, -10.137, -156.835, 56.671, 166.77]
  Set speed (16.5 mm/s)
  Call Extruder(179.17732)
  MoveL 6448 to (529.22, 445.36, 112) mm, rotated rx 180 ry 0 rz 160 deg; joints [-0.68, 64.924, -10.879, -156.583, 56.353, 166.506]
  Set speed (16.5 mm/s)
  Call Extruder(187.04235)
  MoveL 6449 to (531.23, 446.49, 112) mm, rotated rx 180 ry 0 rz 160 deg; joints [-0.543, 65.276, -11.598, -156.325, 56.048, 166.24]
  Set speed (16.5 mm/s)
  Call Extruder(194.76792)
  MoveL 6450 to (533.16, 447.66, 112) mm, rotated rx -180 ry 0 rz 160 deg; joints [-0.402, 65.619, -12.297, -156.061, 55.756, 165.973]
  Set speed (16.5 mm/s)
  Call Extruder(202.64529)
  MoveL 6451 to (535.09, 448.93, 112) mm, rotated rx 180 ry 0 rz 160 deg; joints [-0.25, 65.964, -13.002, -155.782, 55.465, 165.695]
  Set speed (16.5 mm/s)
  Call Extruder(210.07238)
  MoveL 6452 to (536.86, 450.2, 112) mm, rotated rx 180 ry 0 rz 160 deg; joints [-0.1, 66.286, -13.657, -155.511, 55.199, 165.428]
  Set speed (16.5 mm/s)
  Call Extruder(218.22139)
  MoveL 6453 to (538.75, 451.65, 112) mm, rotated rx 180 ry 0 rz 160 deg; joints [0.071, 66.634, -14.365, -155.204, 54.916, 165.129]
  Call Extruder(225.91644)
  MoveL 6454 to (540.48, 453.09, 112) mm, rotated rx 180 ry 0 rz 160 deg; joints [0.24, 66.958, -15.021, -154.906, 54.657, 164.842]
  Set speed (16.5 mm/s)
  Call Extruder(233.81046)
  MoveL 6455 to (542.2, 454.64, 112) mm, rotated rx 180 ry 0 rz 160 deg; joints [0.419, 67.283, -15.682, -154.592, 54.401, 164.544]
  Set speed (16.5 mm/s)
  Call Extruder(241.51181)
  MoveL 6456 to (543.82, 456.2, 112) mm, rotated rx 180 ry 0 rz 160 deg; joints [0.599, 67.595, -16.313, -154.278, 54.162, 164.249]
  Call Extruder(245.73035)
  MoveL 6457 to (544.69, 457.08, 112) mm, rotated rx 180 ry 0 rz 160 deg; joints [0.701, 67.762, -16.652, -154.104, 54.035, 164.086]
  Set speed (16.5 mm/s)
  Call Extruder(250.13576)
  MoveL 6458 to (545.57, 458.02, 112) mm, rotated rx 180 ry 0 rz 160 deg; joints [0.808, 67.935, -17.002, -153.92, 53.905, 163.915]
  Set speed (16.5 mm/s)
  Call Extruder(254.36998)
  MoveL 6459 to (546.4, 458.94, 112) mm, rotated rx 180 ry 0 rz 160 deg; joints [0.913, 68.099, -17.333, -153.741, 53.784, 163.75]
  Set speed (16.5 mm/s)
  Call Extruder(258.17415)
  MoveL 6460 to (547.13, 459.78, 112) mm, rotated rx -180 ry 0 rz 160 deg; joints [1.009, 68.244, -17.627, -153.579, 53.678, 163.601]
  Set speed (16.5 mm/s)
  Call Extruder(262.65166)
  MoveL 6461 to (547.97, 460.79, 112) mm, rotated rx 180 ry 0 rz 160 deg; joints [1.123, 68.413, -17.967, -153.386, 53.557, 163.425]
  Set speed (16.5 mm/s)
  Call Extruder(267.49272)
  MoveL 6462 to (548.86, 461.9, 112) mm, rotated rx 180 ry 0 rz 160 deg; joints [1.248, 68.592, -18.328, -153.176, 53.43, 163.234]
  Call Extruder(271.10839)
  MoveL 6463 to (549.5, 462.74, 112) mm, rotated rx -180 ry 0 rz 160 deg; joints [1.343, 68.723, -18.593, -153.018, 53.338, 163.091]
  Call Extruder(275.98843)
  MoveL 6464 to (550.35, 463.89, 112) mm, rotated rx 180 ry 0 rz 160 deg; joints [1.473, 68.898, -18.946, -152.803, 53.218, 162.898]
  Set speed (16.5 mm/s)
  Call Extruder(280.30865)
  MoveL 6465 to (551.07, 464.92, 112) mm, rotated rx -180 ry 0 rz 160 deg; joints [1.589, 69.049, -19.25, -152.612, 53.116, 162.727]
  Set speed (16.5 mm/s)
  Call Extruder(283.92789)
  MoveL 6466 to (551.67, 465.8, 112) mm, rotated rx -180 ry 0 rz 160 deg; joints [1.688, 69.173, -19.501, -152.45, 53.033, 162.583]
  Set speed (16.5 mm/s)
  Call Extruder(288.43654)
  MoveL 6467 to (552.38, 466.91, 112) mm, rotated rx -180 ry 0 rz 160 deg; joints [1.812, 69.325, -19.807, -152.248, 52.934, 162.404]
  Set speed (16.5 mm/s)
  Call Extruder(292.75019)
  MoveL 6468 to (553.05, 467.99, 112) mm, rotated rx -180 ry 0 rz 160 deg; joints [1.932, 69.467, -20.093, -152.054, 52.844, 162.233]
  Set speed (16.5 mm/s)
  Call Extruder(297.75862)
  MoveL 6469 to (553.79, 469.25, 112) mm, rotated rx 180 ry 0 rz 160 deg; joints [2.073, 69.629, -20.417, -151.827, 52.743, 162.035]
  Set speed (16.5 mm/s)
  Call Extruder(303.77532)
  MoveL 6470 to (554.65, 470.79, 112) mm, rotated rx -180 ry 0 rz 160 deg; joints [2.244, 69.817, -20.796, -151.553, 52.628, 161.797]
  Set speed (16.5 mm/s)
  Call Extruder(310.04787)
  MoveL 6471 to (555.49, 472.43, 112) mm, rotated rx -180 ry 0 rz 160 deg; joints [2.426, 70.005, -21.174, -151.267, 52.519, 161.551]
  Set speed (16.5 mm/s)
  Call Extruder(314.93424)
  MoveL 6472 to (556.11, 473.72, 112) mm, rotated rx -180 ry 0 rz 160 deg; joints [2.569, 70.146, -21.458, -151.043, 52.44, 161.36]
  Set speed (16.5 mm/s)
  Call Extruder(319.21680)
  MoveL 6473 to (556.63, 474.86, 112) mm, rotated rx 180 ry 0 rz 160 deg; joints [2.695, 70.266, -21.698, -150.847, 52.374, 161.194]
  Set speed (16.5 mm/s)
  Call Extruder(323.70566)
  MoveL 6474 to (557.14, 476.06, 112) mm, rotated rx -180 ry 0 rz 160 deg; joints [2.829, 70.387, -21.941, -150.642, 52.311, 161.022]
  Set speed (16.5 mm/s)
  Call Extruder(328.03696)
  MoveL 6475 to (557.63, 477.24, 112) mm, rotated rx -180 ry 0 rz 160 deg; joints [2.958, 70.502, -22.171, -150.443, 52.253, 160.856]
  Set speed (16.5 mm/s)
  Call Extruder(332.37692)
  MoveL 6476 to (558.08, 478.42, 112) mm, rotated rx 180 ry 0 rz 160 deg; joints [3.089, 70.61, -22.389, -150.245, 52.202, 160.691]
  Set speed (16.5 mm/s)
  Call Extruder(336.62020)
  MoveL 6477 to (558.5, 479.59, 112) mm, rotated rx 180 ry 0 rz 160 deg; joints [3.218, 70.714, -22.597, -150.051, 52.154, 160.531]
  Set speed (16.5 mm/s)
  Call Extruder(341.04944)
  MoveL 6478 to (558.91, 480.82, 112) mm, rotated rx -180 ry 0 rz 160 deg; joints [3.353, 70.817, -22.803, -149.849, 52.11, 160.367]
  Set speed (16.5 mm/s)
  Call Extruder(345.32843)
  MoveL 6479 to (559.29, 482.01, 112) mm, rotated rx 180 ry 0 rz 160 deg; joints [3.484, 70.914, -22.997, -149.654, 52.07, 160.208]
  Set speed (16.5 mm/s)
  Call Extruder(349.71439)
  MoveL 6480 to (559.64, 483.24, 112) mm, rotated rx 180 ry 0 rz 160 deg; joints [3.62, 71.006, -23.183, -149.455, 52.036, 160.049]
  Set speed (16.5 mm/s)
  Call Extruder(353.77624)
  MoveL 6481 to (559.96, 484.39, 112) mm, rotated rx -180 ry 0 rz 160 deg; joints [3.746, 71.09, -23.351, -149.271, 52.007, 159.902]
  Call Extruder(358.38204)
  MoveL 6482 to (560.28, 485.7, 112) mm, rotated rx 180 ry 0 rz 160 deg; joints [3.89, 71.179, -23.527, -149.064, 51.981, 159.739]
  Set speed (16.5 mm/s)
  Call Extruder(362.78265)
  MoveL 6483 to (560.57, 486.95, 112) mm, rotated rx -180 ry 0 rz 160 deg; joints [4.028, 71.261, -23.692, -148.867, 51.958, 159.584]
  Set speed (16.5 mm/s)
  Call Extruder(371.39608)
  MoveL 6484 to (561.05, 489.42, 112) mm, rotated rx -180 ry 0 rz 160 deg; joints [4.301, 71.405, -23.981, -148.484, 51.931, 159.289]
  Set speed (16.5 mm/s)
  Call Extruder(380.05125)
  MoveL 6485 to (561.43, 491.93, 112) mm, rotated rx 180 ry 0 rz 160 deg; joints [4.577, 71.531, -24.233, -148.104, 51.922, 159.002]
  Set speed (16.5 mm/s)
  Call Extruder(388.79817)
  MoveL 6486 to (561.71, 494.48, 112) mm, rotated rx -180 ry 0 rz 160 deg; joints [4.858, 71.639, -24.449, -147.726, 51.931, 158.724]
  Set speed (16.5 mm/s)
  Call Extruder(397.36149)
  MoveL 6487 to (561.89, 496.98, 112) mm, rotated rx -180 ry 0 rz 160 deg; joints [5.135, 71.726, -24.622, -147.363, 51.96, 158.464]
  Set speed (16.5 mm/s)
  Call Extruder(406.01794)
  MoveL 6488 to (561.96, 499.51, 112) mm, rotated rx 180 ry 0 rz 160 deg; joints [5.416, 71.794, -24.757, -147.003, 52.006, 158.213]
  Set speed (16.5 mm/s)
  Call Extruder(414.77768)
  MoveL 6489 to (561.92, 502.07, 112) mm, rotated rx -180 ry 0 rz 160 deg; joints [5.701, 71.842, -24.853, -146.647, 52.073, 157.973]
  Set speed (16.5 mm/s)
  Call Extruder(423.32329)
  MoveL 6490 to (561.79, 504.57, 112) mm, rotated rx 180 ry 0 rz 160 deg; joints [5.979, 71.868, -24.907, -146.309, 52.155, 157.754]
  Set speed (16.5 mm/s)
  Call Extruder(431.97513)
  MoveL 6491 to (561.55, 507.1, 112) mm, rotated rx -180 ry 0 rz 160 deg; joints [6.262, 71.876, -24.921, -145.975, 52.257, 157.546]
  Set speed (16.5 mm/s)
  Call Extruder(440.72030)
  MoveL 6492 to (561.21, 509.63, 112) mm, rotated rx 180 ry 0 rz 160 deg; joints [6.547, 71.862, -24.894, -145.648, 52.378, 157.352]
  Set speed (16.5 mm/s)
  Call Extruder(449.29184)
  MoveL 6493 to (560.77, 512.1, 112) mm, rotated rx 180 ry 0 rz 160 deg; joints [6.827, 71.829, -24.828, -145.337, 52.513, 157.178]
  Set speed (16.5 mm/s)
  Call Extruder(457.96046)
  MoveL 6494 to (560.22, 514.58, 112) mm, rotated rx -180 ry 0 rz 160 deg; joints [7.109, 71.775, -24.72, -145.034, 52.667, 157.018]
  Set speed (16.5 mm/s)
  Call Extruder(462.26185)
  MoveL 6495 to (559.91, 515.8, 112) mm, rotated rx -180 ry 0 rz 160 deg; joints [7.248, 71.74, -24.65, -144.888, 52.75, 156.946]
  Call Extruder(466.69088)
  MoveL 6496 to (559.57, 517.05, 112) mm, rotated rx 180 ry 0 rz 160 deg; joints [7.391, 71.701, -24.571, -144.74, 52.838, 156.874]
  Set speed (16.5 mm/s)
  Call Extruder(470.93827)
  MoveL 6497 to (559.21, 518.24, 112) mm, rotated rx -180 ry 0 rz 160 deg; joints [7.528, 71.656, -24.482, -144.601, 52.928, 156.811]
  Call Extruder(475.30256)
  MoveL 6498 to (558.83, 519.46, 112) mm, rotated rx 180 ry 0 rz 160 deg; joints [7.668, 71.608, -24.386, -144.461, 53.023, 156.748]
  Set speed (16.5 mm/s)
  Call Extruder(483.82444)
  MoveL 6499 to (558, 521.81, 112) mm, rotated rx 180 ry 0 rz 160 deg; joints [7.942, 71.496, -24.163, -144.196, 53.221, 156.641]
  Set speed (16.5 mm/s)
  Call Extruder(492.38038)
  MoveL 6500 to (557.07, 524.14, 112) mm, rotated rx 180 ry 0 rz 160 deg; joints [8.214, 71.366, -23.903, -143.941, 53.435, 156.55]
  Set speed (16.5 mm/s)
  Call Extruder(496.91014)
  MoveL 6501 to (556.53, 525.35, 112) mm, rotated rx 180 ry 0 rz 160 deg; joints [8.357, 71.289, -23.748, -143.812, 53.555, 156.51]
  Set speed (16.5 mm/s)
  Call Extruder(501.03319)
  MoveL 6502 to (556.03, 526.45, 112) mm, rotated rx 180 ry 0 rz 160 deg; joints [8.487, 71.216, -23.603, -143.695, 53.665, 156.476]
  Set speed (16.5 mm/s)
  Call Extruder(505.60416)
  MoveL 6503 to (555.45, 527.65, 112) mm, rotated rx 180 ry 0 rz 160 deg; joints [8.63, 71.129, -23.429, -143.57, 53.792, 156.443]
  Set speed (16.5 mm/s)
  Call Extruder(509.75126)
  MoveL 6504 to (554.89, 528.73, 112) mm, rotated rx 180 ry 0 rz 160 deg; joints [8.76, 71.046, -23.262, -143.459, 53.911, 156.418]
  Set speed (16.5 mm/s)
  Call Extruder(514.11289)
  MoveL 6505 to (554.29, 529.86, 112) mm, rotated rx -180 ry 0 rz 160 deg; joints [8.895, 70.955, -23.079, -143.346, 54.039, 156.395]
  Set speed (16.5 mm/s)
  Call Extruder(518.57672)
  MoveL 6506 to (553.65, 531, 112) mm, rotated rx 180 ry 0 rz 160 deg; joints [9.033, 70.857, -22.883, -143.232, 54.173, 156.377]
  Set speed (16.5 mm/s)
  Call Extruder(523.64499)
  MoveL 6507 to (552.89, 532.27, 112) mm, rotated rx 180 ry 0 rz 160 deg; joints [9.188, 70.74, -22.649, -143.108, 54.329, 156.361]
  Set speed (16.5 mm/s)
  Call Extruder(527.23734)
  MoveL 6508 to (552.34, 533.16, 112) mm, rotated rx 180 ry 0 rz 160 deg; joints [9.298, 70.653, -22.475, -143.022, 54.442, 156.353]
  Call Extruder(531.53524)
  MoveL 6509 to (551.65, 534.22, 112) mm, rotated rx -180 ry 0 rz 160 deg; joints [9.428, 70.546, -22.26, -142.922, 54.58, 156.348]
  Set speed (16.5 mm/s)
  Call Extruder(535.85909)
  MoveL 6510 to (550.95, 535.27, 112) mm, rotated rx -180 ry 0 rz 160 deg; joints [9.557, 70.434, -22.036, -142.824, 54.722, 156.347]
  Set speed (16.5 mm/s)
  Call Extruder(540.05213)
  MoveL 6511 to (550.24, 536.27, 112) mm, rotated rx -180 ry 0 rz 160 deg; joints [9.683, 70.322, -21.811, -142.732, 54.862, 156.35]
  Set speed (16.5 mm/s)
  Call Extruder(543.83512)
  MoveL 6512 to (549.58, 537.16, 112) mm, rotated rx -180 ry 0 rz 160 deg; joints [9.795, 70.218, -21.601, -142.652, 54.991, 156.355]
  Call Extruder(548.71514)
  MoveL 6513 to (548.71, 538.3, 112) mm, rotated rx 180 ry 0 rz 160 deg; joints [9.938, 70.079, -21.322, -142.551, 55.159, 156.367]
  Call Extruder(552.49245)
  MoveL 6514 to (548.02, 539.16, 112) mm, rotated rx 180 ry 0 rz 160 deg; joints [10.048, 69.968, -21.1, -142.475, 55.292, 156.38]
  Set speed (16.5 mm/s)
  Call Extruder(556.82547)
  MoveL 6515 to (547.2, 540.13, 112) mm, rotated rx -180 ry 0 rz 160 deg; joints [10.173, 69.838, -20.838, -142.391, 55.447, 156.399]
  Call Extruder(561.19767)
  MoveL 6516 to (546.37, 541.1, 112) mm, rotated rx 180 ry 0 rz 160 deg; joints [10.298, 69.703, -20.567, -142.309, 55.605, 156.421]
  Set speed (16.5 mm/s)
  Call Extruder(568.50452)
  MoveL 6517 to (544.92, 542.68, 112) mm, rotated rx 180 ry 0 rz 160 deg; joints [10.505, 69.47, -20.098, -142.179, 55.873, 156.467]
  Set speed (16.5 mm/s)
  Call Extruder(574.65301)
  MoveL 6518 to (543.66, 543.96, 112) mm, rotated rx 180 ry 0 rz 160 deg; joints [10.675, 69.266, -19.688, -142.076, 56.104, 156.514]
  Set speed (16.5 mm/s)
  Call Extruder(579.05039)
  MoveL 6519 to (542.74, 544.86, 112) mm, rotated rx 180 ry 0 rz 160 deg; joints [10.795, 69.117, -19.387, -142.005, 56.272, 156.552]
  Call Extruder(583.30969)
  MoveL 6520 to (541.83, 545.71, 112) mm, rotated rx 180 ry 0 rz 160 deg; joints [10.911, 68.969, -19.089, -141.939, 56.436, 156.593]
  Set speed (16.5 mm/s)
  Call Extruder(587.72696)
  MoveL 6521 to (540.87, 546.58, 112) mm, rotated rx -180 ry 0 rz 160 deg; joints [11.029, 68.813, -18.774, -141.874, 56.608, 156.638]
  Set speed (16.5 mm/s)
  Call Extruder(591.98766)
  MoveL 6522 to (539.92, 547.39, 112) mm, rotated rx -180 ry 0 rz 160 deg; joints [11.141, 68.659, -18.465, -141.814, 56.775, 156.686]
  Call Extruder(596.46450)
  MoveL 6523 to (538.91, 548.22, 112) mm, rotated rx -180 ry 0 rz 160 deg; joints [11.258, 68.495, -18.134, -141.754, 56.952, 156.739]
  Set speed (16.5 mm/s)
  Call Extruder(601.56274)
  MoveL 6524 to (537.74, 549.14, 112) mm, rotated rx -180 ry 0 rz 160 deg; joints [11.389, 68.305, -17.749, -141.689, 57.156, 156.805]
  Call Extruder(605.10639)
  MoveL 6525 to (536.91, 549.77, 112) mm, rotated rx -180 ry 0 rz 160 deg; joints [11.478, 68.17, -17.478, -141.645, 57.299, 156.853]
  Set speed (16.5 mm/s)
  Call Extruder(609.28248)
  MoveL 6526 to (535.92, 550.49, 112) mm, rotated rx 180 ry 0 rz 160 deg; joints [11.583, 68.01, -17.153, -141.597, 57.469, 156.913]
  Set speed (16.5 mm/s)
  Call Extruder(613.66841)
  MoveL 6527 to (534.87, 551.22, 112) mm, rotated rx 180 ry 0 rz 160 deg; joints [11.69, 67.839, -16.807, -141.548, 57.648, 156.979]
  Set speed (16.5 mm/s)
  Call Extruder(617.44114)
  MoveL 6528 to (533.95, 551.83, 112) mm, rotated rx 180 ry 0 rz 160 deg; joints [11.782, 67.689, -16.505, -141.509, 57.803, 157.038]
  Call Extruder(621.77320)
  MoveL 6529 to (532.88, 552.52, 112) mm, rotated rx 180 ry 0 rz 160 deg; joints [11.885, 67.516, -16.154, -141.466, 57.982, 157.109]
  Set speed (16.5 mm/s)
  Call Extruder(626.75904)
  MoveL 6530 to (531.63, 553.28, 112) mm, rotated rx -180 ry 0 rz 160 deg; joints [12.001, 67.314, -15.744, -141.42, 58.19, 157.194]
  Call Extruder(630.46883)
  MoveL 6531 to (530.69, 553.82, 112) mm, rotated rx 180 ry 0 rz 160 deg; joints [12.087, 67.162, -15.436, -141.388, 58.345, 157.26]
  Set speed (16.5 mm/s)
  Call Extruder(634.75330)
  MoveL 6532 to (529.6, 554.43, 112) mm, rotated rx 180 ry 0 rz 160 deg; joints [12.183, 66.985, -15.077, -141.353, 58.524, 157.339]
  Set speed (16.5 mm/s)
  Call Extruder(640.97478)
  MoveL 6533 to (527.99, 555.28, 112) mm, rotated rx -180 ry 0 rz 160 deg; joints [12.32, 66.725, -14.549, -141.307, 58.786, 157.458]
  Set speed (16.5 mm/s)
  Call Extruder(644.00240)
  MoveL 6534 to (527.19, 555.67, 112) mm, rotated rx -180 ry 0 rz 160 deg; joints [12.385, 66.597, -14.289, -141.287, 58.914, 157.518]
  Set speed (16.5 mm/s)
  Call Extruder(648.49213)
  MoveL 6535 to (526.01, 556.24, 112) mm, rotated rx -180 ry 0 rz 160 deg; joints [12.48, 66.406, -13.9, -141.259, 59.104, 157.609]
  Set speed (16.5 mm/s)
  Call Extruder(652.75882)
  MoveL 6536 to (524.87, 556.75, 112) mm, rotated rx -180 ry 0 rz 160 deg; joints [12.568, 66.222, -13.527, -141.235, 59.286, 157.7]
  Set speed (16.5 mm/s)
  Call Extruder(657.08957)
  MoveL 6537 to (523.71, 557.25, 112) mm, rotated rx 180 ry 0 rz 160 deg; joints [12.655, 66.035, -13.146, -141.213, 59.47, 157.793]
  Set speed (16.5 mm/s)
  Call Extruder(661.42512)
  MoveL 6538 to (522.53, 557.71, 112) mm, rotated rx 180 ry 0 rz 160 deg; joints [12.74, 65.846, -12.76, -141.194, 59.655, 157.889]
  Set speed (16.5 mm/s)
  Call Extruder(665.77802)
  MoveL 6539 to (521.34, 558.17, 112) mm, rotated rx -180 ry 0 rz 160 deg; joints [12.824, 65.656, -12.372, -141.176, 59.841, 157.987]
  Set speed (16.5 mm/s)
  Call Extruder(674.31285)
  MoveL 6540 to (518.98, 558.98, 112) mm, rotated rx -180 ry 0 rz 160 deg; joints [12.981, 65.277, -11.6, -141.151, 60.206, 158.188]
  Set speed (16.5 mm/s)
  Call Extruder(679.70215)
  MoveL 6541 to (517.47, 559.44, 112) mm, rotated rx -180 ry 0 rz 160 deg; joints [13.075, 65.036, -11.108, -141.14, 60.436, 158.32]
  Set speed (16.5 mm/s)
  Call Extruder(682.88842)
  MoveL 6542 to (516.57, 559.7, 112) mm, rotated rx -180 ry 0 rz 160 deg; joints [13.129, 64.894, -10.817, -141.135, 60.573, 158.399]
  Set speed (16.5 mm/s)
  Call Extruder(687.41562)
  MoveL 6543 to (515.29, 560.04, 112) mm, rotated rx 180 ry 0 rz 160 deg; joints [13.204, 64.689, -10.398, -141.131, 60.766, 158.514]
  Set speed (16.5 mm/s)
  Call Extruder(691.80982)
  MoveL 6544 to (514.05, 560.35, 112) mm, rotated rx -180 ry 0 rz 160 deg; joints [13.274, 64.491, -9.992, -141.129, 60.954, 158.627]
  Set speed (16.5 mm/s)
  Call Extruder(700.16674)
  MoveL 6545 to (511.65, 560.85, 112) mm, rotated rx -180 ry 0 rz 160 deg; joints [13.4, 64.111, -9.213, -141.132, 61.31, 158.848]
  Call Extruder(709.18255)
  MoveL 6546 to (509.05, 561.3, 112) mm, rotated rx 180 ry 0 rz 160 deg; joints [13.526, 63.699, -8.367, -141.147, 61.694, 159.094]
  Set speed (16.5 mm/s)
  Call Extruder(717.74983)
  MoveL 6547 to (506.56, 561.61, 112) mm, rotated rx 180 ry 0 rz 160 deg; joints [13.634, 63.306, -7.558, -141.171, 62.056, 159.335]
  Set speed (16.5 mm/s)
  Call Extruder(726.46566)
  MoveL 6548 to (504.02, 561.83, 112) mm, rotated rx 180 ry 0 rz 160 deg; joints [13.734, 62.905, -6.733, -141.206, 62.422, 159.587]
  Set speed (16.5 mm/s)
  Call Extruder(735.16452)
  MoveL 6549 to (501.47, 561.94, 112) mm, rotated rx 180 ry 0 rz 160 deg; joints [13.822, 62.505, -5.908, -141.251, 62.784, 159.844]
  Set speed (16.5 mm/s)
  Call Extruder(743.51975)
  MoveL 6550 to (499.03, 561.95, 112) mm, rotated rx 180 ry 0 rz 160 deg; joints [13.896, 62.122, -5.115, -141.304, 63.129, 160.097]
  Set speed (10.0 mm/s)
  MoveL 6551 to (499.03, 561.95, 116) mm, rotated rx 180 ry 0 rz 160 deg; joints [13.896, 61.504, -4.864, -141.187, 62.842, 159.839]
  Set speed (120.0 mm/s)
  MoveL 6552 to (499.03, 560.11, 116) mm, rotated rx 180 ry 0 rz 160 deg; joints [13.674, 61.434, -4.718, -141.445, 62.824, 159.998]
  Set speed (16.2 mm/s)
  Call Extruder(752.14012)
  MoveL 6553 to (496.55, 560.02, 116) mm, rotated rx -180 ry 0 rz 160 deg; joints [13.736, 61.045, -3.918, -141.51, 63.168, 160.256]
  Set speed (16.2 mm/s)
  Call Extruder(760.72684)
  MoveL 6554 to (494.09, 559.83, 116) mm, rotated rx 180 ry 0 rz 160 deg; joints [13.786, 60.659, -3.122, -141.586, 63.506, 160.518]
  Call Extruder(769.20471)
  MoveL 6555 to (491.67, 559.54, 116) mm, rotated rx -180 ry 0 rz 160 deg; joints [13.823, 60.28, -2.338, -141.671, 63.835, 160.781]
  Set speed (16.2 mm/s)
  Call Extruder(777.63972)
  MoveL 6556 to (489.28, 559.16, 116) mm, rotated rx 180 ry 0 rz 160 deg; joints [13.848, 59.905, -1.563, -141.765, 64.158, 161.045]
  Set speed (16.2 mm/s)
  Call Extruder(786.43460)
  MoveL 6557 to (486.8, 558.65, 116) mm, rotated rx 180 ry 0 rz 160 deg; joints [13.861, 59.517, -0.759, -141.875, 64.489, 161.324]
  Set speed (16.2 mm/s)
  Call Extruder(790.64830)
  MoveL 6558 to (485.63, 558.37, 116) mm, rotated rx -180 ry 0 rz 160 deg; joints [13.863, 59.333, -0.377, -141.932, 64.645, 161.459]
  Set speed (16.2 mm/s)
  Call Extruder(794.73088)
  MoveL 6559 to (484.49, 558.08, 116) mm, rotated rx -180 ry 0 rz 160 deg; joints [13.862, 59.156, -0.009, -141.988, 64.795, 161.59]
  Set speed (16.2 mm/s)
  Call Extruder(799.16634)
  MoveL 6560 to (483.27, 557.74, 116) mm, rotated rx -180 ry 0 rz 160 deg; joints [13.856, 58.964, 0.39, -142.054, 64.957, 161.733]
  Set speed (16.2 mm/s)
  Call Extruder(803.57073)
  MoveL 6561 to (482.05, 557.38, 116) mm, rotated rx 180 ry 0 rz 160 deg; joints [13.849, 58.775, 0.784, -142.12, 65.116, 161.875]
  Set speed (16.2 mm/s)
  Call Extruder(811.88139)
  MoveL 6562 to (479.79, 556.62, 116) mm, rotated rx -180 ry 0 rz 160 deg; joints [13.824, 58.421, 1.521, -142.255, 65.411, 162.145]
  Set speed (16.2 mm/s)
  Call Extruder(816.33961)
  MoveL 6563 to (478.59, 556.17, 116) mm, rotated rx -180 ry 0 rz 160 deg; joints [13.804, 58.233, 1.913, -142.332, 65.567, 162.29]
  Set speed (16.2 mm/s)
  Call Extruder(820.51656)
  MoveL 6564 to (477.47, 555.74, 116) mm, rotated rx -180 ry 0 rz 160 deg; joints [13.784, 58.059, 2.278, -142.405, 65.711, 162.426]
  Set speed (16.2 mm/s)
  Call Extruder(827.20376)
  MoveL 6565 to (475.71, 554.99, 116) mm, rotated rx 180 ry 0 rz 160 deg; joints [13.744, 57.782, 2.855, -142.53, 65.938, 162.645]
  Set speed (16.2 mm/s)
  Call Extruder(833.37046)
  MoveL 6566 to (474.1, 554.25, 116) mm, rotated rx -180 ry 0 rz 160 deg; joints [13.7, 57.531, 3.382, -142.65, 66.144, 162.847]
  Set speed (16.2 mm/s)
  Call Extruder(837.66442)
  MoveL 6567 to (472.99, 553.71, 116) mm, rotated rx -180 ry 0 rz 160 deg; joints [13.665, 57.357, 3.747, -142.737, 66.285, 162.987]
  Set speed (16.2 mm/s)
  Call Extruder(840.77724)
  MoveL 6568 to (472.19, 553.3, 116) mm, rotated rx -180 ry 0 rz 160 deg; joints [13.638, 57.232, 4.008, -142.802, 66.386, 163.089]
  Set speed (16.2 mm/s)
  Call Extruder(846.25726)
  MoveL 6569 to (470.81, 552.56, 116) mm, rotated rx -180 ry 0 rz 160 deg; joints [13.585, 57.015, 4.465, -142.92, 66.561, 163.269]
  Set speed (16.2 mm/s)
  Call Extruder(850.52028)
  MoveL 6570 to (469.75, 551.95, 116) mm, rotated rx 180 ry 0 rz 160 deg; joints [13.54, 56.847, 4.816, -143.016, 66.695, 163.409]
  Set speed (16.2 mm/s)
  Call Extruder(855.45680)
  MoveL 6571 to (468.53, 551.22, 116) mm, rotated rx -180 ry 0 rz 160 deg; joints [13.483, 56.656, 5.219, -143.129, 66.849, 163.57]
  Set speed (16.2 mm/s)
  Call Extruder(859.11724)
  MoveL 6572 to (467.64, 550.66, 116) mm, rotated rx -180 ry 0 rz 160 deg; joints [13.438, 56.516, 5.515, -143.216, 66.96, 163.69]
  Call Extruder(863.42423)
  MoveL 6573 to (466.6, 549.99, 116) mm, rotated rx 180 ry 0 rz 160 deg; joints [13.382, 56.352, 5.859, -143.32, 67.089, 163.83]
  Set speed (16.2 mm/s)
  Call Extruder(867.73107)
  MoveL 6574 to (465.58, 549.29, 116) mm, rotated rx -180 ry 0 rz 160 deg; joints [13.323, 56.191, 6.199, -143.427, 67.216, 163.97]
  Call Extruder(871.88727)
  MoveL 6575 to (464.61, 548.59, 116) mm, rotated rx -180 ry 0 rz 160 deg; joints [13.262, 56.037, 6.524, -143.533, 67.337, 164.104]
  Set speed (16.2 mm/s)
  Call Extruder(876.17863)
  MoveL 6576 to (463.62, 547.86, 116) mm, rotated rx 180 ry 0 rz 160 deg; joints [13.196, 55.881, 6.855, -143.645, 67.459, 164.243]
  Set speed (16.2 mm/s)
  Call Extruder(880.42413)
  MoveL 6577 to (462.65, 547.11, 116) mm, rotated rx 180 ry 0 rz 160 deg; joints [13.127, 55.728, 7.178, -143.758, 67.578, 164.38]
  Set speed (16.2 mm/s)
  Call Extruder(884.85242)
  MoveL 6578 to (461.66, 546.31, 116) mm, rotated rx 180 ry 0 rz 160 deg; joints [13.052, 55.571, 7.511, -143.879, 67.7, 164.522]
  Call Extruder(889.01019)
  MoveL 6579 to (460.75, 545.54, 116) mm, rotated rx -180 ry 0 rz 160 deg; joints [12.978, 55.426, 7.818, -143.996, 67.811, 164.654]
  Set speed (16.2 mm/s)
  Call Extruder(893.30496)
  MoveL 6580 to (459.83, 544.72, 116) mm, rotated rx 180 ry 0 rz 160 deg; joints [12.897, 55.278, 8.132, -144.119, 67.924, 164.791]
  Call Extruder(897.68708)
  MoveL 6581 to (458.89, 543.87, 116) mm, rotated rx 180 ry 0 rz 160 deg; joints [12.813, 55.129, 8.447, -144.247, 68.037, 164.929]
  Set speed (16.2 mm/s)
  Call Extruder(901.83761)
  MoveL 6582 to (458.03, 543.05, 116) mm, rotated rx 180 ry 0 rz 160 deg; joints [12.729, 54.991, 8.741, -144.371, 68.142, 165.059]
  Set speed (16.2 mm/s)
  Call Extruder(906.12663)
  MoveL 6583 to (457.16, 542.18, 116) mm, rotated rx 180 ry 0 rz 160 deg; joints [12.638, 54.851, 9.039, -144.501, 68.247, 165.193]
  Call Extruder(910.37703)
  MoveL 6584 to (456.31, 541.3, 116) mm, rotated rx 180 ry 0 rz 160 deg; joints [12.546, 54.714, 9.33, -144.634, 68.349, 165.325]
  Set speed (16.2 mm/s)
  Call Extruder(914.70695)
  MoveL 6585 to (455.47, 540.39, 116) mm, rotated rx 180 ry 0 rz 160 deg; joints [12.448, 54.578, 9.621, -144.771, 68.451, 165.459]
  Set speed (16.2 mm/s)
  Call Extruder(918.95662)
  MoveL 6586 to (454.66, 539.47, 116) mm, rotated rx -180 ry 0 rz 160 deg; joints [12.348, 54.446, 9.902, -144.908, 68.548, 165.589]
  Set speed (16.2 mm/s)
  Call Extruder(923.21392)
  MoveL 6587 to (453.86, 538.54, 116) mm, rotated rx 180 ry 0 rz 160 deg; joints [12.246, 54.317, 10.177, -145.048, 68.642, 165.718]
  Set speed (16.2 mm/s)
  Call Extruder(926.09102)
  MoveL 6588 to (453.34, 537.9, 116) mm, rotated rx -180 ry 0 rz 160 deg; joints [12.175, 54.231, 10.361, -145.144, 68.705, 165.805]
  Call Extruder(931.74744)
  MoveL 6589 to (452.33, 536.63, 116) mm, rotated rx 180 ry 0 rz 160 deg; joints [12.03, 54.066, 10.714, -145.336, 68.824, 165.975]
  Set speed (16.2 mm/s)
  Call Extruder(936.09808)
  MoveL 6590 to (451.58, 535.63, 116) mm, rotated rx -180 ry 0 rz 160 deg; joints [11.915, 53.942, 10.978, -145.486, 68.912, 166.103]
  Set speed (16.2 mm/s)
  Call Extruder(940.28921)
  MoveL 6591 to (450.87, 534.65, 116) mm, rotated rx 180 ry 0 rz 160 deg; joints [11.801, 53.825, 11.228, -145.633, 68.995, 166.226]
  Set speed (16.2 mm/s)
  Call Extruder(945.32634)
  MoveL 6592 to (450.05, 533.46, 116) mm, rotated rx -180 ry 0 rz 160 deg; joints [11.661, 53.689, 11.521, -145.813, 69.091, 166.373]
  Set speed (16.2 mm/s)
  Call Extruder(949.01014)
  MoveL 6593 to (449.47, 532.57, 116) mm, rotated rx -180 ry 0 rz 160 deg; joints [11.556, 53.592, 11.729, -145.947, 69.158, 166.479]
  Set speed (16.2 mm/s)
  Call Extruder(953.13935)
  MoveL 6594 to (448.84, 531.57, 116) mm, rotated rx 180 ry 0 rz 160 deg; joints [11.435, 53.485, 11.958, -146.098, 69.231, 166.596]
  Set speed (16.2 mm/s)
  Call Extruder(957.46382)
  MoveL 6595 to (448.19, 530.5, 116) mm, rotated rx -180 ry 0 rz 160 deg; joints [11.305, 53.377, 12.191, -146.259, 69.304, 166.718]
  Set speed (16.2 mm/s)
  Call Extruder(961.74082)
  MoveL 6596 to (447.58, 529.44, 116) mm, rotated rx -180 ry 0 rz 160 deg; joints [11.174, 53.272, 12.415, -146.42, 69.374, 166.837]
  Set speed (16.2 mm/s)
  Call Extruder(966.03825)
  MoveL 6597 to (446.99, 528.36, 116) mm, rotated rx 180 ry 0 rz 160 deg; joints [11.04, 53.171, 12.633, -146.584, 69.441, 166.955]
  Set speed (16.2 mm/s)
  Call Extruder(970.29076)
  MoveL 6598 to (446.42, 527.27, 116) mm, rotated rx -180 ry 0 rz 160 deg; joints [10.904, 53.073, 12.844, -146.749, 69.505, 167.071]
  Set speed (16.2 mm/s)
  Call Extruder(974.52076)
  MoveL 6599 to (445.88, 526.19, 116) mm, rotated rx 180 ry 0 rz 160 deg; joints [10.767, 52.979, 13.046, -146.914, 69.565, 167.184]
  Set speed (16.2 mm/s)
  Call Extruder(978.97365)
  MoveL 6600 to (445.34, 525.03, 116) mm, rotated rx 180 ry 0 rz 160 deg; joints [10.618, 52.884, 13.251, -147.091, 69.625, 167.302]
  Set speed (16.2 mm/s)
  Call Extruder(983.15145)
  MoveL 6601 to (444.85, 523.93, 116) mm, rotated rx -180 ry 0 rz 160 deg; joints [10.478, 52.797, 13.44, -147.257, 69.679, 167.411]
  Call Extruder(987.53130)
  MoveL 6602 to (444.37, 522.77, 116) mm, rotated rx -180 ry 0 rz 160 deg; joints [10.327, 52.71, 13.627, -147.434, 69.731, 167.524]
  Set speed (16.2 mm/s)
  Call Extruder(991.98656)
  MoveL 6603 to (443.89, 521.59, 116) mm, rotated rx 180 ry 0 rz 160 deg; joints [10.172, 52.624, 13.813, -147.616, 69.782, 167.637]
  Set speed (16.2 mm/s)
  Call Extruder(996.11228)
  MoveL 6604 to (443.48, 520.48, 116) mm, rotated rx -180 ry 0 rz 160 deg; joints [10.025, 52.548, 13.977, -147.786, 69.825, 167.74]
  Call Extruder(1000.51864)
  MoveL 6605 to (443.06, 519.28, 116) mm, rotated rx -180 ry 0 rz 160 deg; joints [9.867, 52.47, 14.146, -147.968, 69.868, 167.848]
  Set speed (16.2 mm/s)
  Call Extruder(1008.95896)
  MoveL 6606 to (442.33, 516.97, 116) mm, rotated rx -180 ry 0 rz 160 deg; joints [9.556, 52.33, 14.449, -148.323, 69.942, 168.051]
  Set speed (16.2 mm/s)
  Call Extruder(1017.33916)
  MoveL 6607 to (441.69, 514.65, 116) mm, rotated rx -180 ry 0 rz 160 deg; joints [9.24, 52.204, 14.722, -148.68, 70.002, 168.245]
  Call Extruder(1025.78413)
  MoveL 6608 to (441.15, 512.28, 116) mm, rotated rx 180 ry 0 rz 160 deg; joints [8.914, 52.09, 14.968, -149.045, 70.05, 168.434]
  Set speed (16.2 mm/s)
  Call Extruder(1034.66314)
  MoveL 6609 to (440.68, 509.78, 116) mm, rotated rx -180 ry 0 rz 160 deg; joints [8.565, 51.985, 15.196, -149.432, 70.086, 168.625]
  Set speed (16.2 mm/s)
  Call Extruder(1043.20873)
  MoveL 6610 to (440.33, 507.35, 116) mm, rotated rx 180 ry 0 rz 160 deg; joints [8.223, 51.898, 15.386, -149.807, 70.107, 168.802]
  Call Extruder(1051.76623)
  MoveL 6611 to (440.08, 504.9, 116) mm, rotated rx 180 ry 0 rz 160 deg; joints [7.875, 51.825, 15.545, -150.186, 70.115, 168.971]
  Set speed (16.2 mm/s)
  Call Extruder(1060.13745)
  MoveL 6612 to (439.93, 502.5, 116) mm, rotated rx -180 ry 0 rz 160 deg; joints [7.531, 51.767, 15.671, -150.557, 70.108, 169.129]
  Set speed (16.2 mm/s)
  Call Extruder(1068.78895)
  MoveL 6613 to (439.88, 500.01, 116) mm, rotated rx 180 ry 0 rz 160 deg; joints [7.172, 51.721, 15.77, -150.942, 70.088, 169.284]
  Set speed (16.2 mm/s)
  Call Extruder(1076.58187)
  MoveL 6614 to (439.92, 497.77, 116) mm, rotated rx -180 ry 0 rz 160 deg; joints [6.846, 51.692, 15.833, -151.288, 70.057, 169.417]
  Set speed (16.2 mm/s)
  Call Extruder(1084.18102)
  MoveL 6615 to (440.04, 495.59, 116) mm, rotated rx -180 ry 0 rz 160 deg; joints [6.528, 51.676, 15.869, -151.624, 70.016, 169.541]
  Set speed (16.2 mm/s)
  Call Extruder(1091.88367)
  MoveL 6616 to (440.25, 493.39, 116) mm, rotated rx 180 ry 0 rz 160 deg; joints [6.204, 51.67, 15.881, -151.964, 69.964, 169.66]
  Call Extruder(1099.57616)
  MoveL 6617 to (440.53, 491.2, 116) mm, rotated rx 180 ry 0 rz 160 deg; joints [5.881, 51.677, 15.867, -152.302, 69.899, 169.773]
  Set speed (16.2 mm/s)
  Call Extruder(1107.37447)
  MoveL 6618 to (440.9, 488.99, 116) mm, rotated rx -180 ry 0 rz 160 deg; joints [5.554, 51.695, 15.827, -152.641, 69.822, 169.88]
  Set speed (16.2 mm/s)
  Call Extruder(1114.98554)
  MoveL 6619 to (441.34, 486.84, 116) mm, rotated rx -180 ry 0 rz 160 deg; joints [5.236, 51.724, 15.763, -152.968, 69.736, 169.979]
  Call Extruder(1122.69378)
  MoveL 6620 to (441.86, 484.69, 116) mm, rotated rx -180 ry 0 rz 160 deg; joints [4.917, 51.765, 15.674, -153.296, 69.638, 170.072]
  Set speed (16.2 mm/s)
  Call Extruder(1130.39833)
  MoveL 6621 to (442.47, 482.56, 116) mm, rotated rx 180 ry 0 rz 160 deg; joints [4.6, 51.818, 15.56, -153.619, 69.528, 170.159]
  Call Extruder(1138.09743)
  MoveL 6622 to (443.15, 480.46, 116) mm, rotated rx -180 ry 0 rz 160 deg; joints [4.286, 51.882, 15.421, -153.936, 69.408, 170.239]
  Set speed (16.2 mm/s)
  Call Extruder(1145.83587)
  MoveL 6623 to (443.91, 478.37, 116) mm, rotated rx -180 ry 0 rz 160 deg; joints [3.975, 51.957, 15.256, -154.249, 69.275, 170.313]
  Set speed (16.2 mm/s)
  Call Extruder(1152.66106)
  MoveL 6624 to (444.64, 476.55, 116) mm, rotated rx 180 ry 0 rz 160 deg; joints [3.704, 52.033, 15.091, -154.52, 69.149, 170.373]
  Set speed (16.2 mm/s)
  Call Extruder(1161.11121)
  MoveL 6625 to (445.64, 474.33, 116) mm, rotated rx 180 ry 0 rz 160 deg; joints [3.375, 52.14, 14.86, -154.847, 68.982, 170.44]
  Set speed (16.2 mm/s)
  Call Extruder(1169.00162)
  MoveL 6626 to (446.64, 472.3, 116) mm, rotated rx -180 ry 0 rz 160 deg; joints [3.074, 52.251, 14.618, -155.145, 68.814, 170.496]
  Call Extruder(1176.51009)
  MoveL 6627 to (447.67, 470.4, 116) mm, rotated rx -180 ry 0 rz 160 deg; joints [2.792, 52.368, 14.366, -155.421, 68.644, 170.543]
  Set speed (16.2 mm/s)
  Call Extruder(1184.35130)
  MoveL 6628 to (448.82, 468.46, 116) mm, rotated rx -180 ry 0 rz 160 deg; joints [2.506, 52.501, 14.078, -155.699, 68.456, 170.586]
  Set speed (16.2 mm/s)
  Call Extruder(1192.00592)
  MoveL 6629 to (450.01, 466.61, 116) mm, rotated rx 180 ry 0 rz 160 deg; joints [2.233, 52.641, 13.775, -155.962, 68.263, 170.621]
  Set speed (16.2 mm/s)
  Call Extruder(1199.70745)
  MoveL 6630 to (451.27, 464.79, 116) mm, rotated rx 180 ry 0 rz 160 deg; joints [1.966, 52.793, 13.447, -156.217, 68.059, 170.649]
  Call Extruder(1207.45104)
  MoveL 6631 to (452.61, 463.01, 116) mm, rotated rx 180 ry 0 rz 160 deg; joints [1.706, 52.956, 13.096, -156.464, 67.844, 170.672]
  Call Extruder(1215.15276)
  MoveL 6632 to (454, 461.29, 116) mm, rotated rx -180 ry 0 rz 160 deg; joints [1.456, 53.128, 12.725, -156.698, 67.621, 170.687]
  Set speed (16.2 mm/s)
  Call Extruder(1222.80980)
  MoveL 6633 to (455.45, 459.63, 116) mm, rotated rx 180 ry 0 rz 160 deg; joints [1.216, 53.309, 12.335, -156.92, 67.391, 170.697]
  Set speed (16.2 mm/s)
  Call Extruder(1230.43366)
  MoveL 6634 to (456.95, 458.04, 116) mm, rotated rx 180 ry 0 rz 160 deg; joints [0.987, 53.5, 11.927, -157.13, 67.153, 170.699]
  Call Extruder(1238.06654)
  MoveL 6635 to (458.51, 456.5, 116) mm, rotated rx -180 ry 0 rz 160 deg; joints [0.766, 53.699, 11.499, -157.329, 66.906, 170.695]
  Call Extruder(1245.89333)
  MoveL 6636 to (460.17, 454.97, 116) mm, rotated rx 180 ry 0 rz 160 deg; joints [0.55, 53.913, 11.04, -157.521, 66.646, 170.684]
  Set speed (16.2 mm/s)
  Call Extruder(1253.39836)
  MoveL 6637 to (461.81, 453.57, 116) mm, rotated rx -180 ry 0 rz 160 deg; joints [0.353, 54.128, 10.582, -157.692, 66.388, 170.668]
  Set speed (16.2 mm/s)
  Call Extruder(1261.75933)
  MoveL 6638 to (463.69, 452.08, 116) mm, rotated rx -180 ry 0 rz 160 deg; joints [0.144, 54.376, 10.051, -157.87, 66.093, 170.642]
  Set speed (16.2 mm/s)
  Call Extruder(1268.49208)
  MoveL 6639 to (465.25, 450.94, 116) mm, rotated rx 180 ry 0 rz 160 deg; joints [-0.014, 54.583, 9.609, -158.002, 65.85, 170.615]
  Set speed (16.2 mm/s)
  Call Extruder(1276.75615)
  MoveL 6640 to (467.22, 449.61, 116) mm, rotated rx 180 ry 0 rz 160 deg; joints [-0.197, 54.846, 9.048, -158.15, 65.544, 170.575]
  Set speed (16.2 mm/s)
  Call Extruder(1284.50538)
  MoveL 6641 to (469.1, 448.43, 116) mm, rotated rx 180 ry 0 rz 160 deg; joints [-0.358, 55.102, 8.506, -158.276, 65.25, 170.53]
  Set speed (16.2 mm/s)
  Call Extruder(1292.19542)
  MoveL 6642 to (471.02, 447.33, 116) mm, rotated rx 180 ry 0 rz 160 deg; joints [-0.506, 55.363, 7.951, -158.387, 64.954, 170.478]
  Set speed (16.2 mm/s)
  Call Extruder(1299.85269)
  MoveL 6643 to (472.97, 446.3, 116) mm, rotated rx -180 ry 0 rz 160 deg; joints [-0.643, 55.63, 7.385, -158.484, 64.652, 170.42]
  Set speed (16.2 mm/s)
  Call Extruder(1307.56182)
  MoveL 6644 to (474.96, 445.34, 116) mm, rotated rx 180 ry 0 rz 160 deg; joints [-0.77, 55.907, 6.799, -158.568, 64.344, 170.355]
  Call Extruder(1315.31310)
  MoveL 6645 to (477.01, 444.45, 116) mm, rotated rx 180 ry 0 rz 160 deg; joints [-0.886, 56.192, 6.198, -158.639, 64.029, 170.281]
  Set speed (16.2 mm/s)
  Call Extruder(1322.82731)
  MoveL 6646 to (479.02, 443.66, 116) mm, rotated rx -180 ry 0 rz 160 deg; joints [-0.987, 56.475, 5.601, -158.695, 63.72, 170.203]
  Set speed (16.2 mm/s)
  Call Extruder(1330.71639)
  MoveL 6647 to (481.15, 442.91, 116) mm, rotated rx -180 ry 0 rz 160 deg; joints [-1.082, 56.778, 4.963, -158.739, 63.392, 170.114]
  Set speed (16.2 mm/s)
  Call Extruder(1338.35810)
  MoveL 6648 to (483.25, 442.26, 116) mm, rotated rx -180 ry 0 rz 160 deg; joints [-1.163, 57.077, 4.333, -158.768, 63.07, 170.02]
  Set speed (16.2 mm/s)
  Call Extruder(1346.02321)
  MoveL 6649 to (485.38, 441.69, 116) mm, rotated rx -180 ry 0 rz 160 deg; joints [-1.233, 57.384, 3.69, -158.783, 62.744, 169.919]
  Set speed (16.2 mm/s)
  Call Extruder(1353.82438)
  MoveL 6650 to (487.56, 441.18, 116) mm, rotated rx -180 ry 0 rz 160 deg; joints [-1.293, 57.701, 3.026, -158.784, 62.41, 169.808]
  Set speed (16.2 mm/s)
  Call Extruder(1361.33587)
  MoveL 6651 to (489.68, 440.77, 116) mm, rotated rx 180 ry 0 rz 160 deg; joints [-1.34, 58.011, 2.377, -158.772, 62.086, 169.694]
  Set speed (16.2 mm/s)
  Call Extruder(1368.79534)
  MoveL 6652 to (491.8, 440.44, 116) mm, rotated rx 180 ry 0 rz 160 deg; joints [-1.377, 58.323, 1.725, -158.747, 61.762, 169.573]
  Set speed (16.2 mm/s)
  Call Extruder(1376.83434)
  MoveL 6653 to (494.09, 440.17, 116) mm, rotated rx -180 ry 0 rz 160 deg; joints [-1.404, 58.664, 1.014, -158.705, 61.412, 169.435]
  Set speed (16.2 mm/s)
  Call Extruder(1384.56549)
  MoveL 6654 to (496.31, 440, 116) mm, rotated rx -180 ry 0 rz 160 deg; joints [-1.42, 58.996, 0.323, -158.652, 61.075, 169.295]
  Call Extruder(1392.33770)
  MoveL 6655 to (498.54, 439.9, 116) mm, rotated rx -180 ry 0 rz 160 deg; joints [-1.425, 59.334, -0.378, -158.584, 60.735, 169.146]
  Set speed (16.2 mm/s)
  Call Extruder(1399.95758)
  MoveL 6656 to (500.73, 439.89, 116) mm, rotated rx 180 ry 0 rz 160 deg; joints [-1.42, 59.668, -1.071, -158.504, 60.402, 168.992]
  Set speed (16.2 mm/s)
  Call Extruder(1407.73534)
  MoveL 6657 to (502.96, 439.95, 116) mm, rotated rx 180 ry 0 rz 160 deg; joints [-1.405, 60.012, -1.784, -158.409, 60.062, 168.828]
  Set speed (16.2 mm/s)
  Call Extruder(1415.34193)
  MoveL 6658 to (505.15, 440.1, 116) mm, rotated rx 180 ry 0 rz 160 deg; joints [-1.379, 60.35, -2.485, -158.302, 59.731, 168.659]
  Set speed (16.2 mm/s)
  Call Extruder(1422.86950)
  MoveL 6659 to (507.3, 440.33, 116) mm, rotated rx 180 ry 0 rz 160 deg; joints [-1.344, 60.687, -3.18, -158.185, 59.405, 168.485]
  Set speed (16.2 mm/s)
  Call Extruder(1430.65467)
  MoveL 6660 to (509.51, 440.64, 116) mm, rotated rx -180 ry 0 rz 160 deg; joints [-1.299, 61.037, -3.902, -158.05, 59.069, 168.297]
  Set speed (16.2 mm/s)
  Call Extruder(1438.43580)
  MoveL 6661 to (511.71, 441.03, 116) mm, rotated rx 180 ry 0 rz 160 deg; joints [-1.244, 61.388, -4.625, -157.903, 58.735, 168.101]
  Set speed (16.2 mm/s)
  Call Extruder(1445.56007)
  MoveL 6662 to (513.72, 441.47, 116) mm, rotated rx 180 ry 0 rz 160 deg; joints [-1.185, 61.71, -5.287, -157.758, 58.432, 167.916]
  Set speed (16.2 mm/s)
  Call Extruder(1453.75805)
  MoveL 6663 to (516, 442.05, 116) mm, rotated rx 180 ry 0 rz 160 deg; joints [-1.108, 62.081, -6.048, -157.577, 58.087, 167.695]
  Set speed (16.2 mm/s)
  Call Extruder(1461.40472)
  MoveL 6664 to (518.1, 442.67, 116) mm, rotated rx 180 ry 0 rz 160 deg; joints [-1.026, 62.427, -6.758, -157.395, 57.769, 167.48]
  Call Extruder(1469.33873)
  MoveL 6665 to (520.26, 443.4, 116) mm, rotated rx 180 ry 0 rz 160 deg; joints [-0.932, 62.785, -7.492, -157.195, 57.443, 167.251]
  Call Extruder(1476.95102)
  MoveL 6666 to (522.31, 444.18, 116) mm, rotated rx 180 ry 0 rz 160 deg; joints [-0.834, 63.128, -8.193, -156.992, 57.135, 167.024]
  Set speed (16.2 mm/s)
  Call Extruder(1484.75661)
  MoveL 6667 to (524.38, 445.05, 116) mm, rotated rx 180 ry 0 rz 160 deg; joints [-0.725, 63.478, -8.908, -156.772, 56.824, 166.784]
  Call Extruder(1492.44942)
  MoveL 6668 to (526.38, 445.98, 116) mm, rotated rx 180 ry 0 rz 160 deg; joints [-0.61, 63.822, -9.609, -156.545, 56.523, 166.541]
  Set speed (16.2 mm/s)
  Call Extruder(1500.05867)
  MoveL 6669 to (528.33, 446.98, 116) mm, rotated rx 180 ry 0 rz 160 deg; joints [-0.488, 64.159, -10.295, -156.31, 56.231, 166.294]
  Set speed (16.2 mm/s)
  Call Extruder(1507.86491)
  MoveL 6670 to (530.29, 448.07, 116) mm, rotated rx -180 ry 0 rz 160 deg; joints [-0.355, 64.502, -10.993, -156.058, 55.938, 166.035]
  Set speed (16.2 mm/s)
  Call Extruder(1515.44924)
  MoveL 6671 to (532.15, 449.2, 116) mm, rotated rx -180 ry 0 rz 160 deg; joints [-0.219, 64.832, -11.664, -155.804, 55.66, 165.777]
  Set speed (16.2 mm/s)
  Call Extruder(1523.25467)
  MoveL 6672 to (534.02, 450.44, 116) mm, rotated rx 180 ry 0 rz 160 deg; joints [-0.072, 65.167, -12.345, -155.533, 55.382, 165.506]
  Set speed (16.2 mm/s)
  Call Extruder(1530.86354)
  MoveL 6673 to (535.8, 451.7, 116) mm, rotated rx -180 ry 0 rz 160 deg; joints [0.078, 65.491, -13, -155.261, 55.118, 165.237]
  Set speed (16.2 mm/s)
  Call Extruder(1538.43596)
  MoveL 6674 to (537.53, 453.03, 116) mm, rotated rx -180 ry 0 rz 160 deg; joints [0.234, 65.808, -13.642, -154.981, 54.863, 164.965]
  Set speed (16.2 mm/s)
  Call Extruder(1546.25723)
  MoveL 6675 to (539.26, 454.47, 116) mm, rotated rx 180 ry 0 rz 160 deg; joints [0.402, 66.13, -14.293, -154.684, 54.609, 164.679]
  Set speed (16.2 mm/s)
  Call Extruder(1554.21305)
  MoveL 6676 to (540.96, 456, 116) mm, rotated rx 180 ry 0 rz 160 deg; joints [0.579, 66.451, -14.942, -154.373, 54.361, 164.384]
  Set speed (16.2 mm/s)
  Call Extruder(1561.70710)
  MoveL 6677 to (542.51, 457.49, 116) mm, rotated rx 180 ry 0 rz 160 deg; joints [0.751, 66.747, -15.54, -154.074, 54.136, 164.103]
  Set speed (16.2 mm/s)
  Call Extruder(1565.90919)
  MoveL 6678 to (543.36, 458.35, 116) mm, rotated rx -180 ry 0 rz 160 deg; joints [0.85, 66.911, -15.87, -153.904, 54.013, 163.944]
  Set speed (16.2 mm/s)
  Call Extruder(1570.15113)
  MoveL 6679 to (544.19, 459.24, 116) mm, rotated rx -180 ry 0 rz 160 deg; joints [0.952, 67.073, -16.198, -153.73, 53.894, 163.783]
  Call Extruder(0.00000)
  Set speed (16.2 mm/s)
  Call Extruder(4.30184)
  MoveL 6680 to (545.02, 460.16, 116) mm, rotated rx -180 ry 0 rz 160 deg; joints [1.057, 67.236, -16.526, -153.552, 53.775, 163.618]
  Set speed (16.2 mm/s)
  Call Extruder(8.55428)
  MoveL 6681 to (545.82, 461.08, 116) mm, rotated rx 180 ry 0 rz 160 deg; joints [1.162, 67.394, -16.845, -153.374, 53.661, 163.455]
  Set speed (16.2 mm/s)
  Call Extruder(12.91767)
  MoveL 6682 to (546.62, 462.05, 116) mm, rotated rx -180 ry 0 rz 160 deg; joints [1.271, 67.555, -17.168, -153.19, 53.547, 163.287]
  Set speed (16.2 mm/s)
  Call Extruder(17.20176)
  MoveL 6683 to (547.39, 463.01, 116) mm, rotated rx -180 ry 0 rz 160 deg; joints [1.38, 67.709, -17.479, -153.008, 53.439, 163.122]
  Set speed (16.2 mm/s)
  Call Extruder(21.46830)
  MoveL 6684 to (548.14, 463.98, 116) mm, rotated rx 180 ry 0 rz 160 deg; joints [1.49, 67.861, -17.783, -152.825, 53.335, 162.957]
  Set speed (16.2 mm/s)
  Call Extruder(25.63690)
  MoveL 6685 to (548.84, 464.95, 116) mm, rotated rx -180 ry 0 rz 160 deg; joints [1.599, 68.006, -18.075, -152.645, 53.237, 162.795]
  Set speed (16.2 mm/s)
  Call Extruder(29.93335)
  MoveL 6686 to (549.55, 465.96, 116) mm, rotated rx 180 ry 0 rz 160 deg; joints [1.713, 68.152, -18.369, -152.458, 53.139, 162.629]
  Set speed (16.2 mm/s)
  Call Extruder(34.34130)
  MoveL 6687 to (550.26, 467.01, 116) mm, rotated rx 180 ry 0 rz 160 deg; joints [1.831, 68.3, -18.666, -152.266, 53.043, 162.458]
  Set speed (16.2 mm/s)
  Call Extruder(38.52921)
  MoveL 6688 to (550.91, 468.02, 116) mm, rotated rx -180 ry 0 rz 160 deg; joints [1.944, 68.437, -18.942, -152.082, 52.955, 162.296]
  Set speed (16.2 mm/s)
  Call Extruder(42.78631)
  MoveL 6689 to (551.55, 469.07, 116) mm, rotated rx 180 ry 0 rz 160 deg; joints [2.061, 68.573, -19.215, -151.894, 52.87, 162.131]
  Set speed (16.2 mm/s)
  Call Extruder(47.07953)
  MoveL 6690 to (552.17, 470.13, 116) mm, rotated rx -180 ry 0 rz 160 deg; joints [2.18, 68.708, -19.484, -151.704, 52.787, 161.965]
  Set speed (16.2 mm/s)
  Call Extruder(53.69957)
  MoveL 6691 to (553.1, 471.8, 116) mm, rotated rx 180 ry 0 rz 160 deg; joints [2.366, 68.91, -19.888, -151.408, 52.667, 161.71]
  Set speed (16.2 mm/s)
  Call Extruder(59.85952)
  MoveL 6692 to (553.9, 473.38, 116) mm, rotated rx -180 ry 0 rz 160 deg; joints [2.541, 69.089, -20.247, -151.133, 52.565, 161.474]
  Set speed (16.2 mm/s)
  Call Extruder(64.22788)
  MoveL 6693 to (554.44, 474.51, 116) mm, rotated rx 180 ry 0 rz 160 deg; joints [2.667, 69.211, -20.492, -150.937, 52.498, 161.307]
  Call Extruder(68.53893)
  MoveL 6694 to (554.96, 475.63, 116) mm, rotated rx 180 ry 0 rz 160 deg; joints [2.792, 69.329, -20.728, -150.744, 52.435, 161.144]
  Set speed (16.2 mm/s)
  Call Extruder(77.01940)
  MoveL 6695 to (555.9, 477.88, 116) mm, rotated rx -180 ry 0 rz 160 deg; joints [3.041, 69.549, -21.169, -150.363, 52.324, 160.826]
  Set speed (16.2 mm/s)
  Call Extruder(81.39324)
  MoveL 6696 to (556.35, 479.06, 116) mm, rotated rx 180 ry 0 rz 160 deg; joints [3.171, 69.655, -21.381, -150.167, 52.275, 160.664]
  Set speed (16.2 mm/s)
  Call Extruder(85.44417)
  MoveL 6697 to (556.74, 480.15, 116) mm, rotated rx -180 ry 0 rz 160 deg; joints [3.292, 69.752, -21.574, -149.985, 52.231, 160.515]
  Set speed (16.2 mm/s)
  Call Extruder(89.93692)
  MoveL 6698 to (557.15, 481.37, 116) mm, rotated rx -180 ry 0 rz 160 deg; joints [3.427, 69.853, -21.776, -149.785, 52.189, 160.352]
  Set speed (16.2 mm/s)
  Call Extruder(94.13745)
  MoveL 6699 to (557.52, 482.52, 116) mm, rotated rx 180 ry 0 rz 160 deg; joints [3.554, 69.946, -21.962, -149.598, 52.152, 160.2]
  Set speed (16.2 mm/s)
  Call Extruder(102.54725)
  MoveL 6700 to (558.18, 484.84, 116) mm, rotated rx -180 ry 0 rz 160 deg; joints [3.811, 70.117, -22.304, -149.224, 52.092, 159.902]
  Set speed (16.2 mm/s)
  Call Extruder(111.32558)
  MoveL 6701 to (558.76, 487.3, 116) mm, rotated rx -180 ry 0 rz 160 deg; joints [4.082, 70.279, -22.627, -148.837, 52.048, 159.599]
  Set speed (16.2 mm/s)
  Call Extruder(119.86144)
  MoveL 6702 to (559.23, 489.71, 116) mm, rotated rx -180 ry 0 rz 160 deg; joints [4.348, 70.417, -22.903, -148.465, 52.024, 159.314]
  Call Extruder(128.33210)
  MoveL 6703 to (559.6, 492.11, 116) mm, rotated rx 180 ry 0 rz 160 deg; joints [4.614, 70.538, -23.143, -148.1, 52.016, 159.04]
  Set speed (16.2 mm/s)
  Call Extruder(137.09133)
  MoveL 6704 to (559.88, 494.61, 116) mm, rotated rx 180 ry 0 rz 160 deg; joints [4.891, 70.643, -23.354, -147.729, 52.027, 158.767]
  Set speed (16.2 mm/s)
  Call Extruder(145.54070)
  MoveL 6705 to (560.05, 497.04, 116) mm, rotated rx -180 ry 0 rz 160 deg; joints [5.16, 70.726, -23.52, -147.377, 52.055, 158.515]
  Call Extruder(154.09828)
  MoveL 6706 to (560.12, 499.5, 116) mm, rotated rx 180 ry 0 rz 160 deg; joints [5.434, 70.791, -23.649, -147.027, 52.102, 158.273]
  Set speed (16.2 mm/s)
  Call Extruder(162.49450)
  MoveL 6707 to (560.09, 501.91, 116) mm, rotated rx -180 ry 0 rz 160 deg; joints [5.703, 70.836, -23.739, -146.692, 52.164, 158.048]
  Set speed (16.2 mm/s)
  Call Extruder(171.19971)
  MoveL 6708 to (559.96, 504.41, 116) mm, rotated rx 180 ry 0 rz 160 deg; joints [5.982, 70.863, -23.793, -146.352, 52.247, 157.828]
  Call Extruder(179.63401)
  MoveL 6709 to (559.73, 506.82, 116) mm, rotated rx -180 ry 0 rz 160 deg; joints [6.254, 70.871, -23.807, -146.032, 52.344, 157.629]
  Call Extruder(188.41035)
  MoveL 6710 to (559.39, 509.32, 116) mm, rotated rx 180 ry 0 rz 160 deg; joints [6.536, 70.858, -23.782, -145.708, 52.462, 157.437]
  Set speed (16.2 mm/s)
  Call Extruder(196.75057)
  MoveL 6711 to (558.97, 511.68, 116) mm, rotated rx 180 ry 0 rz 160 deg; joints [6.804, 70.826, -23.719, -145.41, 52.591, 157.27]
  Set speed (16.2 mm/s)
  Call Extruder(205.22175)
  MoveL 6712 to (558.45, 514.06, 116) mm, rotated rx -180 ry 0 rz 160 deg; joints [7.075, 70.776, -23.618, -145.117, 52.738, 157.115]
  Set speed (16.2 mm/s)
  Call Extruder(209.73126)
  MoveL 6713 to (558.13, 515.32, 116) mm, rotated rx -180 ry 0 rz 160 deg; joints [7.219, 70.74, -23.548, -144.966, 52.822, 157.039]
  Set speed (16.2 mm/s)
  Call Extruder(214.20840)
  MoveL 6714 to (557.79, 516.56, 116) mm, rotated rx -180 ry 0 rz 160 deg; joints [7.362, 70.702, -23.472, -144.818, 52.909, 156.967]
  Set speed (16.2 mm/s)
  Call Extruder(222.56114)
  MoveL 6715 to (557.09, 518.85, 116) mm, rotated rx 180 ry 0 rz 160 deg; joints [7.627, 70.615, -23.297, -144.55, 53.084, 156.847]
  Call Extruder(231.07717)
  MoveL 6716 to (556.27, 521.16, 116) mm, rotated rx -180 ry 0 rz 160 deg; joints [7.896, 70.507, -23.082, -144.288, 53.277, 156.739]
  Set speed (16.2 mm/s)
  Call Extruder(235.42050)
  MoveL 6717 to (555.82, 522.32, 116) mm, rotated rx 180 ry 0 rz 160 deg; joints [8.032, 70.444, -22.957, -144.159, 53.382, 156.692]
  Call Extruder(239.45652)
  MoveL 6718 to (555.38, 523.39, 116) mm, rotated rx 180 ry 0 rz 160 deg; joints [8.158, 70.384, -22.836, -144.041, 53.481, 156.65]
  Call Extruder(243.97448)
  MoveL 6719 to (554.86, 524.58, 116) mm, rotated rx -180 ry 0 rz 160 deg; joints [8.299, 70.309, -22.687, -143.913, 53.597, 156.609]
  Set speed (16.2 mm/s)
  Call Extruder(248.17094)
  MoveL 6720 to (554.36, 525.68, 116) mm, rotated rx 180 ry 0 rz 160 deg; joints [8.429, 70.237, -22.544, -143.796, 53.706, 156.573]
  Set speed (16.2 mm/s)
  Call Extruder(251.37373)
  MoveL 6721 to (553.96, 526.51, 116) mm, rotated rx 180 ry 0 rz 160 deg; joints [8.528, 70.179, -22.428, -143.708, 53.792, 156.549]
  Set speed (16.2 mm/s)
  Call Extruder(258.84351)
  MoveL 6722 to (552.98, 528.42, 116) mm, rotated rx -180 ry 0 rz 160 deg; joints [8.758, 70.034, -22.137, -143.51, 54, 156.502]
  Set speed (16.2 mm/s)
  Call Extruder(265.26884)
  MoveL 6723 to (552.08, 530.03, 116) mm, rotated rx -180 ry 0 rz 160 deg; joints [8.953, 69.896, -21.863, -143.348, 54.188, 156.473]
  Set speed (16.2 mm/s)
  Call Extruder(269.52223)
  MoveL 6724 to (551.46, 531.08, 116) mm, rotated rx -180 ry 0 rz 160 deg; joints [9.082, 69.802, -21.674, -143.244, 54.315, 156.458]
  Set speed (16.2 mm/s)
  Call Extruder(273.85867)
  MoveL 6725 to (550.8, 532.14, 116) mm, rotated rx -180 ry 0 rz 160 deg; joints [9.212, 69.7, -21.472, -143.14, 54.448, 156.447]
  Set speed (16.2 mm/s)
  Call Extruder(277.46948)
  MoveL 6726 to (550.24, 533.02, 116) mm, rotated rx -180 ry 0 rz 160 deg; joints [9.319, 69.613, -21.298, -143.056, 54.561, 156.441]
  Set speed (16.2 mm/s)
  Call Extruder(282.35697)
  MoveL 6727 to (549.46, 534.18, 116) mm, rotated rx 180 ry 0 rz 160 deg; joints [9.464, 69.491, -21.053, -142.946, 54.716, 156.437]
  Set speed (16.2 mm/s)
  Call Extruder(286.71553)
  MoveL 6728 to (548.73, 535.2, 116) mm, rotated rx 180 ry 0 rz 160 deg; joints [9.592, 69.378, -20.826, -142.851, 54.858, 156.438]
  Call Extruder(290.99171)
  MoveL 6729 to (548, 536.19, 116) mm, rotated rx 180 ry 0 rz 160 deg; joints [9.716, 69.262, -20.595, -142.761, 55, 156.443]
  Call Extruder(295.17615)
  MoveL 6730 to (547.27, 537.15, 116) mm, rotated rx 180 ry 0 rz 160 deg; joints [9.837, 69.147, -20.364, -142.674, 55.14, 156.451]
  Call Extruder(299.50200)
  MoveL 6731 to (546.49, 538.12, 116) mm, rotated rx 180 ry 0 rz 160 deg; joints [9.961, 69.023, -20.116, -142.588, 55.288, 156.464]
  Set speed (16.2 mm/s)
  Call Extruder(303.81996)
  MoveL 6732 to (545.7, 539.07, 116) mm, rotated rx -180 ry 0 rz 160 deg; joints [10.084, 68.896, -19.862, -142.505, 55.438, 156.481]
  Set speed (16.2 mm/s)
  Call Extruder(308.03100)
  MoveL 6733 to (544.9, 539.98, 116) mm, rotated rx 180 ry 0 rz 160 deg; joints [10.202, 68.769, -19.607, -142.427, 55.587, 156.5]
  Set speed (16.2 mm/s)
  Call Extruder(312.43367)
  MoveL 6734 to (544.05, 540.92, 116) mm, rotated rx -180 ry 0 rz 160 deg; joints [10.325, 68.633, -19.334, -142.348, 55.744, 156.525]
  Set speed (16.2 mm/s)
  Call Extruder(315.68333)
  MoveL 6735 to (543.41, 541.6, 116) mm, rotated rx 180 ry 0 rz 160 deg; joints [10.414, 68.53, -19.128, -142.291, 55.862, 156.545]
  Call Extruder(320.86689)
  MoveL 6736 to (542.36, 542.66, 116) mm, rotated rx 180 ry 0 rz 160 deg; joints [10.556, 68.362, -18.791, -142.205, 56.052, 156.583]
  Set speed (16.2 mm/s)
  Call Extruder(325.16041)
  MoveL 6737 to (541.48, 543.52, 116) mm, rotated rx -180 ry 0 rz 160 deg; joints [10.671, 68.22, -18.505, -142.136, 56.211, 156.617]
  Set speed (16.2 mm/s)
  Call Extruder(329.44059)
  MoveL 6738 to (540.58, 544.36, 116) mm, rotated rx 180 ry 0 rz 160 deg; joints [10.785, 68.075, -18.214, -142.07, 56.371, 156.656]
  Set speed (16.2 mm/s)
  Call Extruder(333.74993)
  MoveL 6739 to (539.66, 545.18, 116) mm, rotated rx -180 ry 0 rz 160 deg; joints [10.898, 67.926, -17.915, -142.007, 56.535, 156.698]
  Call Extruder(337.99065)
  MoveL 6740 to (538.73, 545.98, 116) mm, rotated rx -180 ry 0 rz 160 deg; joints [11.008, 67.777, -17.615, -141.947, 56.697, 156.742]
  Set speed (16.2 mm/s)
  Call Extruder(342.31854)
  MoveL 6741 to (537.77, 546.77, 116) mm, rotated rx -180 ry 0 rz 160 deg; joints [11.119, 67.623, -17.304, -141.888, 56.864, 156.791]
  Set speed (16.2 mm/s)
  Call Extruder(346.53839)
  MoveL 6742 to (536.82, 547.52, 116) mm, rotated rx 180 ry 0 rz 160 deg; joints [11.226, 67.469, -16.995, -141.834, 57.028, 156.842]
  Set speed (16.2 mm/s)
  Call Extruder(350.84159)
  MoveL 6743 to (535.84, 548.27, 116) mm, rotated rx -180 ry 0 rz 160 deg; joints [11.333, 67.31, -16.674, -141.781, 57.197, 156.897]
  Set speed (16.2 mm/s)
  Call Extruder(355.16420)
  MoveL 6744 to (534.83, 549, 116) mm, rotated rx 180 ry 0 rz 160 deg; joints [11.439, 67.147, -16.347, -141.731, 57.368, 156.955]
  Set speed (16.2 mm/s)
  Call Extruder(359.40150)
  MoveL 6745 to (533.83, 549.69, 116) mm, rotated rx 180 ry 0 rz 160 deg; joints [11.541, 66.986, -16.021, -141.684, 57.536, 157.016]
  Set speed (16.2 mm/s)
  Call Extruder(363.65362)
  MoveL 6746 to (532.82, 550.37, 116) mm, rotated rx -180 ry 0 rz 160 deg; joints [11.642, 66.822, -15.691, -141.64, 57.707, 157.079]
  Set speed (16.2 mm/s)
  Call Extruder(367.99237)
  MoveL 6747 to (531.76, 551.04, 116) mm, rotated rx -180 ry 0 rz 160 deg; joints [11.743, 66.651, -15.347, -141.598, 57.882, 157.148]
  Set speed (16.2 mm/s)
  Call Extruder(372.26707)
  MoveL 6748 to (530.72, 551.68, 116) mm, rotated rx 180 ry 0 rz 160 deg; joints [11.841, 66.482, -15.005, -141.558, 58.055, 157.218]
  Set speed (16.2 mm/s)
  Call Extruder(376.50164)
  MoveL 6749 to (529.66, 552.29, 116) mm, rotated rx 180 ry 0 rz 160 deg; joints [11.937, 66.312, -14.663, -141.521, 58.227, 157.29]
  Set speed (16.2 mm/s)
  Call Extruder(380.18416)
  MoveL 6750 to (528.74, 552.81, 116) mm, rotated rx -180 ry 0 rz 160 deg; joints [12.018, 66.163, -14.362, -141.491, 58.378, 157.355]
  Set speed (16.2 mm/s)
  Call Extruder(386.39536)
  MoveL 6751 to (527.16, 553.63, 116) mm, rotated rx -180 ry 0 rz 160 deg; joints [12.152, 65.909, -13.847, -141.446, 58.633, 157.469]
  Set speed (16.2 mm/s)
  Call Extruder(389.35081)
  MoveL 6752 to (526.4, 554.01, 116) mm, rotated rx -180 ry 0 rz 160 deg; joints [12.214, 65.786, -13.599, -141.426, 58.755, 157.526]
  Set speed (16.2 mm/s)
  Call Extruder(393.79402)
  MoveL 6753 to (525.25, 554.56, 116) mm, rotated rx 180 ry 0 rz 160 deg; joints [12.306, 65.601, -13.223, -141.398, 58.938, 157.613]
  Set speed (16.2 mm/s)
  Call Extruder(398.01322)
  MoveL 6754 to (524.14, 555.05, 116) mm, rotated rx 180 ry 0 rz 160 deg; joints [12.391, 65.423, -12.863, -141.375, 59.113, 157.699]
  Set speed (16.2 mm/s)
  Call Extruder(402.17007)
  MoveL 6755 to (523.05, 555.53, 116) mm, rotated rx 180 ry 0 rz 160 deg; joints [12.473, 65.247, -12.507, -141.353, 59.285, 157.784]
  Set speed (16.2 mm/s)
  Call Extruder(406.57941)
  MoveL 6756 to (521.87, 555.99, 116) mm, rotated rx -180 ry 0 rz 160 deg; joints [12.558, 65.058, -12.124, -141.334, 59.469, 157.879]
  Set speed (16.2 mm/s)
  Call Extruder(410.91511)
  MoveL 6757 to (520.71, 556.44, 116) mm, rotated rx 180 ry 0 rz 160 deg; joints [12.64, 64.873, -11.746, -141.317, 59.649, 157.973]
  Set speed (16.2 mm/s)
  Call Extruder(415.19467)
  MoveL 6758 to (519.55, 556.85, 116) mm, rotated rx -180 ry 0 rz 160 deg; joints [12.717, 64.687, -11.368, -141.304, 59.828, 158.07]
  Set speed (16.2 mm/s)
  Call Extruder(419.30127)
  MoveL 6759 to (518.43, 557.22, 116) mm, rotated rx -180 ry 0 rz 160 deg; joints [12.79, 64.508, -11.006, -141.292, 59.999, 158.164]
  Call Extruder(423.75076)
  MoveL 6760 to (517.21, 557.6, 116) mm, rotated rx 180 ry 0 rz 160 deg; joints [12.866, 64.313, -10.609, -141.283, 60.185, 158.269]
  Call Extruder(427.84013)
  MoveL 6761 to (516.08, 557.93, 116) mm, rotated rx -180 ry 0 rz 160 deg; joints [12.935, 64.133, -10.243, -141.276, 60.355, 158.366]
  Set speed (16.2 mm/s)
  Call Extruder(430.08085)
  MoveL 6762 to (515.46, 558.1, 116) mm, rotated rx -180 ry 0 rz 160 deg; joints [12.972, 64.035, -10.042, -141.273, 60.448, 158.421]
  Call Extruder(436.44125)
  MoveL 6763 to (513.69, 558.54, 116) mm, rotated rx 180 ry 0 rz 160 deg; joints [13.071, 63.753, -9.468, -141.27, 60.713, 158.578]
  Set speed (16.2 mm/s)
  Call Extruder(445.11477)
  MoveL 6764 to (511.26, 559.06, 116) mm, rotated rx 180 ry 0 rz 160 deg; joints [13.199, 63.365, -8.677, -141.274, 61.074, 158.801]
  Call Extruder(453.75181)
  MoveL 6765 to (508.81, 559.47, 116) mm, rotated rx 180 ry 0 rz 160 deg; joints [13.316, 62.977, -7.884, -141.288, 61.432, 159.03]
  Set speed (16.2 mm/s)
  Call Extruder(462.22505)
  MoveL 6766 to (506.39, 559.78, 116) mm, rotated rx 180 ry 0 rz 160 deg; joints [13.421, 62.595, -7.102, -141.312, 61.782, 159.261]
  Call Extruder(470.83665)
  MoveL 6767 to (503.93, 559.99, 116) mm, rotated rx -180 ry 0 rz 160 deg; joints [13.517, 62.205, -6.304, -141.347, 62.134, 159.502]
  Call Extruder(479.43556)
  MoveL 6768 to (501.46, 560.1, 116) mm, rotated rx -180 ry 0 rz 160 deg; joints [13.602, 61.816, -5.505, -141.391, 62.484, 159.749]
  Set speed (16.2 mm/s)
  Call Extruder(487.89733)
  MoveL 6769 to (499.03, 560.11, 116) mm, rotated rx 180 ry 0 rz 160 deg; joints [13.674, 61.434, -4.718, -141.445, 62.824, 159.998]
  Set speed (10.0 mm/s)
  MoveL 6770 to (499.03, 560.11, 120) mm, rotated rx 180 ry 0 rz 160 deg; joints [13.674, 60.821, -4.48, -141.324, 62.532, 159.735]
  Set speed (120.0 mm/s)
  MoveL 6771 to (499.06, 558.15, 120) mm, rotated rx -180 ry 0 rz 160 deg; joints [13.436, 60.751, -4.338, -141.599, 62.506, 159.902]
  Set speed (16.1 mm/s)
  Call Extruder(496.27366)
  MoveL 6772 to (496.67, 558.06, 120) mm, rotated rx 180 ry 0 rz 160 deg; joints [13.495, 60.374, -3.566, -141.664, 62.836, 160.15]
  Call Extruder(504.63459)
  MoveL 6773 to (494.29, 557.88, 120) mm, rotated rx -180 ry 0 rz 160 deg; joints [13.542, 59.998, -2.796, -141.739, 63.161, 160.401]
  Set speed (16.1 mm/s)
  Call Extruder(512.88780)
  MoveL 6774 to (491.94, 557.6, 120) mm, rotated rx 180 ry 0 rz 160 deg; joints [13.577, 59.63, -2.039, -141.822, 63.478, 160.653]
  Set speed (16.1 mm/s)
  Call Extruder(521.16277)
  MoveL 6775 to (489.61, 557.22, 120) mm, rotated rx -180 ry 0 rz 160 deg; joints [13.6, 59.262, -1.283, -141.917, 63.791, 160.91]
  Call Extruder(529.63579)
  MoveL 6776 to (487.23, 556.74, 120) mm, rotated rx 180 ry 0 rz 160 deg; joints [13.612, 58.888, -0.514, -142.024, 64.107, 161.176]
  Set speed (16.1 mm/s)
  Call Extruder(537.89309)
  MoveL 6777 to (484.94, 556.17, 120) mm, rotated rx -180 ry 0 rz 160 deg; joints [13.61, 58.528, 0.229, -142.138, 64.408, 161.438]
  Set speed (16.1 mm/s)
  Call Extruder(546.09547)
  MoveL 6778 to (482.69, 555.52, 120) mm, rotated rx 180 ry 0 rz 160 deg; joints [13.597, 58.174, 0.96, -142.263, 64.702, 161.7]
  Set speed (16.1 mm/s)
  Call Extruder(554.61965)
  MoveL 6779 to (480.38, 554.75, 120) mm, rotated rx -180 ry 0 rz 160 deg; joints [13.57, 57.81, 1.712, -142.402, 65.001, 161.974]
  Set speed (16.1 mm/s)
  Call Extruder(558.69855)
  MoveL 6780 to (479.29, 554.34, 120) mm, rotated rx 180 ry 0 rz 160 deg; joints [13.551, 57.638, 2.068, -142.474, 65.141, 162.106]
  Set speed (16.1 mm/s)
  Call Extruder(563.10122)
  MoveL 6781 to (478.12, 553.89, 120) mm, rotated rx 180 ry 0 rz 160 deg; joints [13.529, 57.454, 2.451, -142.553, 65.291, 162.248]
  Set speed (16.1 mm/s)
  Call Extruder(570.06950)
  MoveL 6782 to (476.29, 553.11, 120) mm, rotated rx -180 ry 0 rz 160 deg; joints [13.486, 57.165, 3.05, -142.684, 65.525, 162.474]
  Set speed (16.1 mm/s)
  Call Extruder(575.21693)
  MoveL 6783 to (474.95, 552.49, 120) mm, rotated rx -180 ry 0 rz 160 deg; joints [13.448, 56.955, 3.487, -142.786, 65.694, 162.642]
  Set speed (16.1 mm/s)
  Call Extruder(579.42456)
  MoveL 6784 to (473.87, 551.96, 120) mm, rotated rx 180 ry 0 rz 160 deg; joints [13.414, 56.784, 3.842, -142.873, 65.831, 162.778]
  Set speed (16.1 mm/s)
  Call Extruder(581.64331)
  MoveL 6785 to (473.31, 551.66, 120) mm, rotated rx 180 ry 0 rz 160 deg; joints [13.393, 56.695, 4.027, -142.92, 65.901, 162.851]
  Set speed (16.1 mm/s)
  Call Extruder(582.63999)
  MoveL 6786 to (473.05, 551.54, 120) mm, rotated rx 180 ry 0 rz 160 deg; joints [13.385, 56.655, 4.111, -142.94, 65.934, 162.883]
  Set speed (16.1 mm/s)
  Call Extruder(587.70166)
  MoveL 6787 to (471.78, 550.85, 120) mm, rotated rx 180 ry 0 rz 160 deg; joints [13.335, 56.453, 4.53, -143.05, 66.093, 163.048]
  Set speed (16.1 mm/s)
  Call Extruder(592.69148)
  MoveL 6788 to (470.54, 550.15, 120) mm, rotated rx 180 ry 0 rz 160 deg; joints [13.282, 56.257, 4.939, -143.163, 66.248, 163.21]
  Call Extruder(596.07568)
  MoveL 6789 to (469.71, 549.65, 120) mm, rotated rx -180 ry 0 rz 160 deg; joints [13.243, 56.126, 5.213, -143.241, 66.351, 163.32]
  Set speed (16.1 mm/s)
  Call Extruder(600.25018)
  MoveL 6790 to (468.7, 549.02, 120) mm, rotated rx -180 ry 0 rz 160 deg; joints [13.192, 55.965, 5.549, -143.34, 66.476, 163.455]
  Set speed (16.1 mm/s)
  Call Extruder(604.32454)
  MoveL 6791 to (467.73, 548.38, 120) mm, rotated rx 180 ry 0 rz 160 deg; joints [13.139, 55.81, 5.873, -143.439, 66.597, 163.587]
  Set speed (16.1 mm/s)
  Call Extruder(608.61423)
  MoveL 6792 to (466.71, 547.69, 120) mm, rotated rx 180 ry 0 rz 160 deg; joints [13.079, 55.649, 6.21, -143.547, 66.721, 163.726]
  Set speed (16.1 mm/s)
  Call Extruder(612.70498)
  MoveL 6793 to (465.76, 547.01, 120) mm, rotated rx -180 ry 0 rz 160 deg; joints [13.019, 55.497, 6.528, -143.651, 66.838, 163.857]
  Set speed (16.1 mm/s)
  Call Extruder(616.88383)
  MoveL 6794 to (464.8, 546.3, 120) mm, rotated rx 180 ry 0 rz 160 deg; joints [12.955, 55.344, 6.848, -143.761, 66.955, 163.992]
  Set speed (16.1 mm/s)
  Call Extruder(620.98621)
  MoveL 6795 to (463.88, 545.58, 120) mm, rotated rx 180 ry 0 rz 160 deg; joints [12.888, 55.196, 7.159, -143.872, 67.068, 164.123]
  Set speed (16.1 mm/s)
  Call Extruder(625.21060)
  MoveL 6796 to (462.94, 544.82, 120) mm, rotated rx 180 ry 0 rz 160 deg; joints [12.816, 55.045, 7.475, -143.988, 67.182, 164.258]
  Set speed (16.1 mm/s)
  Call Extruder(629.45987)
  MoveL 6797 to (462.01, 544.03, 120) mm, rotated rx 180 ry 0 rz 160 deg; joints [12.74, 54.896, 7.788, -144.108, 67.294, 164.393]
  Set speed (16.1 mm/s)
  Call Extruder(633.53904)
  MoveL 6798 to (461.13, 543.26, 120) mm, rotated rx -180 ry 0 rz 160 deg; joints [12.664, 54.755, 8.084, -144.225, 67.4, 164.522]
  Set speed (16.1 mm/s)
  Call Extruder(637.78677)
  MoveL 6799 to (460.24, 542.44, 120) mm, rotated rx -180 ry 0 rz 160 deg; joints [12.582, 54.611, 8.388, -144.35, 67.507, 164.656]
  Call Extruder(641.85573)
